this is a decoder for a DCF77 signal.
the decoder decodes the DCF77 signal and checks for a valid Date_Time.
since the dcf77 signal is only secured with a simple parity the decoder waits for two consecutive valid transmissions before it sets the output signals.
given a valid reception by the receiver the decoder can take up to 3 minutes to start its clocks the first time.
after a valid signal is detected the error output goes low and dignals a valid dcf signal from the receiver.
a tp is only valid for one program cycle to allow for external rtc setting.
after a valid signal is detected two independent internal clocks are started (RTC and RTC1), the seconds  of these clocks are generated by software since the dcf signal is only valid for minutes.
rtc is always utc ( world time) and rtc1 can be set to any time zone by setting the time_zone_offset and enabling dst for automatic summertime.
a sync output signals the the rtc and rtc1 are in sync with the dcf77 signal, if the dcf77 signal is lost for more then the sync time the sync output goes low
but the rtc and rtc1 outputs keep running based on software timing until a valid dcf77 signal is received again and triggers the clock.
in addition a millisecond output gives further resolutionof the clocks.
a dst output shows if daylight saving time is enables and the weekday output shows which day of week currently is ( 1= monday ... 7= sunday).


*)
(* if tp was set it should only be active for 1 cycle *)
TP := FALSE;

(* read system time *)
t1 := DWORD_TO_TIME(T_PLC_MS());
tx := t1 - last;

IF rec XOR edge THEN
	edge := rec;
	IF NOT rec AND tx > t#1700ms AND tx < t#2000ms THEN
		(* start condition reached *)
		state := 0;
		tp := NOT error;
	ELSIF NOT rec AND tx > t#700ms AND tx < t#1000ms THEN
		(* second switch detected *)
		IF state < 58 THEN state := state +1; ELSE state := 0; END_IF;
	ELSIF rec AND tx  < t#120ms THEN
		(* bit 0 detected  *)
		bits[state] := 0;
	ELSIF rec AND tx > t#120ms AND tx < t#250ms THEN
		(* bit 1 detected *)
		bits[state] := 1;
	ELSE
		(* error condition received signal is not valid *)
		error := TRUE;
		state := 0;
	END_IF;
	last := last + tx;
	IF rec AND state = 58 THEN
		error := FALSE;

		(* decode the bits and check for possible errors *)
		IF bits[0] OR NOT (bits[17] XOR bits[18]) OR NOT bits[20] THEN error := TRUE; END_IF;
		(* decode minute *)
		minute := 0;
		minute.0 := bits[21];
		minute.1 := bits[22];
		minute.2 := bits[23];
		minute.3 := bits[24];
		IF bits[25] THEN minute := minute + 10; END_IF;
		IF bits[26] THEN minute := minute +20; END_IF;
		IF bits[27] THEN minute := minute +40; END_IF;
		IF minute > 59 OR (bits[21] XOR bits[22] XOR bits[23] XOR bits[24] XOR bits[25] XOR bits[26] XOR bits[27] XOR bits[28]) THEN error := TRUE; END_IF;

		(* decode hour *)
		hour := 0;
		hour.0 := bits[29];
		hour.1 := bits[30];
		hour.2 := bits[31];
		hour.3 := bits[32];
		IF bits[33] THEN hour := hour + 10; END_IF;
		IF bits[34] THEN hour := hour +20; END_IF;
		IF hour > 23 OR (bits[29] XOR bits[30] XOR bits[31] XOR bits[32] XOR bits[33] XOR bits[34] XOR bits[35]) THEN error := TRUE; END_IF;

		(* decode day of month *)
		day := 0;
		day.0 := bits[36];
		day.1 := bits[37];
		day.2 := bits[38];
		day.3 := bits[39];
		IF bits[40] THEN day := day + 10; END_IF;
		IF bits[41] THEN day := day + 20; END_IF;
		IF day > 31 THEN error := TRUE; END_IF;

		(* decode day of week *)
		weekday := 0;
		weekday.0 := bits[42];
		weekday.1 := bits[43];
		weekday.2 := bits[44];
		IF weekday > 7 OR weekday < 1 THEN error := TRUE; END_IF;

		(* decode month *)
		month := 0;
		month.0 := bits[45];
		month.1 := bits[46];
		month.2 := bits[47];
		month.3 := bits[48];
		IF bits[49] THEN month := month +10; END_IF;
		IF month > 12 THEN error := TRUE; END_IF;

		(* decode year *)
		year := 0;
		year.0 := bits[50];
		year.1 := bits[51];
		year.2 := bits[52];
		year.3 := bits[53];
		IF bits[54] THEN year := year + 10; END_IF;
		IF bits[55] THEN year := year + 20; END_IF;
		IF bits[56] THEN year := year + 40; END_IF;
		IF bits[57] THEN year := year + 80; END_IF;

		(* check parity for bits 36 to 58 *)
		cnt := 0;
		FOR i := 36 TO 58 DO IF bits[i] THEN cnt := cnt + 1; END_IF; END_FOR;
		IF NOT even(cnt) THEN error := TRUE; END_IF;

		(* time must be valid for two cycles to clear error flag *)
		IF NOT error THEN
			(* set outputs *)
			old_time := mez;
			IF year >= 70 THEN year := year + 1900; ELSE year := year + 2000; END_IF;
			mez := set_DT(year,month,day,hour,minute,0);
			DST := bits[17];
			IF DST THEN
				UTC := DWORD_TO_DT(DT_TO_DWORD(mez) - 7200);
			ELSE
				UTC := DWORD_TO_DT(DT_TO_DWORD(mez) - 3600);
			END_IF

			(* set trigger signal only if the receiver has received 2 successive minutes *)
			IF mez <> old_time + t#1m THEN error := TRUE ; END_IF;
		END_IF;
	END_IF;
END_IF;

(* this portion implements a free running clock which is triggered by the dcf77 signal *)
IF tp THEN
	rtc := utc;
	IF DST AND dst_en THEN
		IF time_offset < 0 THEN	rtc1 := rtc - INT_TO_TIME(-time_offset) + t#1h; ELSE rtc1 := rtc + INT_TO_TIME(time_offset) + t#1h; END_IF;
	ELSE
		IF time_offset < 0 THEN rtc1 := rtc - INT_TO_TIME(-time_offset); ELSE rtc1 := rtc + INT_TO_TIME(time_offset); END_IF;
	END_IF;
	sync := TRUE;
	last_sync := last;
	ty := last;
ELSIF rtc > DWORD_TO_DT(0) AND T1 - ty >= t#1s THEN
	rtc := rtc + t#1s;
	rtc1 := rtc1 + t#1s;
	ty := ty + t#1s;
	sync := ty - last_sync < sync_timeout AND last_sync > DWORD_TO_TIME(0);
	weekday := weekday(DT_TO_DATE(rtc1));
	DST := dst_en AND DST(utc);
END_IF;
msec := TIME_TO_INT(t1 - ty);



(* decode information
bits		content
0			Bitwert immer 0
1 bis 14	reserviert für Betriebsinformationen (nicht für DCF77-Nutzer bestimmt)
15			Rufbit für Alarmierung der PTB-Mitarbeiter
			(bis Mai 2003: Bitwert = 0 falls normale Antenne in Verwendung; 1 = Backupantenne)
16			Bitwert = 1 falls ein Wechsel von MEZ nach MESZ oder umgekehrt bevorsteht; Dauer der Anzeige: 1 Stunde
17 + 18	gültige Zeit = MEZ, falls Bit 17=0 und Bit 18=1
			gültige Zeit = MESZ, falls Bit 17=1 und Bit 18=0
19			Bitwert = 1 falls innerhalb den nächsten 59 Minuten eine Schaltsekunde angeordnet ist. Beim Einfügen einer Schaltsekunde wird anstelle der 59. die 60. Sekundenmarke weggelassen und in der 58. erfolgt ausnahmsweise ein Trägerabfall.
20			Startbit für Zeitinformation (immer 1)
21 - 27		1, 2, 4, 8, 10, 20, 40 Minuten (bitweise Addition)
28			Prüfbit (gerade Parität) für die Bits 21-27
29 - 34		1, 2, 4, 8, 10, 20 Stunden (bitweise Addition)
35			Prüfbit (gerade Parität) für die Bits 29-34
36 - 41		Tagesnummer im aktuellen Monat: 1, 2, 4, 8, 10, 20 (bitweise Addition)
42 - 44		Tagesnummer in der aktuellen Woche: 1, 2, 4 (bitweise Addition)
45 - 49		Monatsnummer: 1, 2, 4, 8, 10 (bitweise Addition)
50 - 57		Jahr (zweistellig): 1, 2, 4, 8, 10, 20, 40, 80 (bitweise Addition)
58			Prüfbit (gerade Parität) füR die Bits 36-57

*)
(* revision history

hm 2.feb 2007		rev 1.1
	change wday and dst outputs when there is no dcf reception

hm	26.feb 2007		rev 1.2
	changed statements where t#1h would be substracted from DT.
	under certain conditions the compiler would crash translating this statement

hm	17. sep 2007	rev 1.3
	replaced time() with T_PLC_MS() for compatibility reasons

hm	24. oct 2007	rev 1.4
	changed dst calculation because function dst was upgraded no error in DCF77 only a change in DST

hm	12. nov 2007	rev 1.5
	changed time_offset from time to integer to allow for negative offset time zones

*)
END_FUNCTION_BLOCK

(* POU Time&Date/DST, ST *)
FUNCTION DST : BOOL
VAR_INPUT
	utc : DT;
END_VAR
VAR
	yr : INT;
	yr4 : DWORD;
	ltc: DWORD;
	idate : DWORD;
END_VAR

(*
version 1.1	24 oct 2007
programmer 	hugo
tested by		tobias

this functions returns TRUE IF dst TIME is active 
the FUNCTION calculates automatically for any year betweek 1970 AND 2099 
wheather daylight savings is on OR off 
the summertime calculation is done according to european standards.
dst will become TRUE AT 01:00 utc in the morning FOR the respective days 
AND it will become FALSE after daylight savings TIME is switched back end OF october at 01:00 utc

*)
yr := year(DT_TO_DATE(utc));
ltc := DT_TO_DWORD(utc);
idate := DT_TO_DWORD(set_DT(yr,3,31,1,0,0));
yr4 := 5*yr/4;
IF idate - ((yr4+4) MOD 7)*86400 <= ltc AND idate + (214 - (yr4+1) MOD 7)*86400 > ltc THEN DST := TRUE; ELSE DST := FALSE; END_IF;

(* revision history
hm	4. aug 2006		rev 1.0
	original version

hm	24. okt 2007	rev 1.1
	deleted time_zone_offset input because dst is generally at 01:00 utc and not mesz
	uk starts 01:00 utc and also greece

*)

(*
Equation used TO calculate the beginning OF European Summer TIME:
Sunday (31 - (5*y/4 + 4) mod 7) March at 01.00 UTC
(valid through 2099, courtesy of Robert H. van Gent, EC).

European Summer Time ends (clocks go back) at 01.00 UTC on

    * 29 October 2006
    * 28 October 2007
    * 26 October 2008

Equation used to calculate the end of European Summer Time:
Sunday (31 - (5*y/4 + 1) mod 7) October at 01.00 UTC
(validity AND credits as above).

*)
END_FUNCTION

(* POU engineering/control/dead_zone, ST *)
FUNCTION dead_zone : REAL
VAR_INPUT
	X : REAL;
	L : REAL;
END_VAR
VAR
END_VAR

(*
version 1.0	12 Feb 2007
programmer 	hugo
tested by		tobias

dead_zone2 is a linear transfer function which follows a linear function except for x is close to 0.
Y = X if abs(x) > L otherwise its 0.

*)
IF ABS(x) > L THEN
	dead_zone := X;
ELSE
	dead_zone := 0;
END_IF;
END_FUNCTION

(* POU engineering/control/dead_zone2, ST *)
FUNCTION_BLOCK dead_zone2
VAR_INPUT
	X : REAL;
	L : REAL;
END_VAR
VAR_OUTPUT
	Y: REAL;
END_VAR
VAR
END_VAR

(*
version 1.0	12 Feb 2007
programmer 	hugo
tested by		tobias

dead_zone2 is a linear transfer function which follows a linear function except for x is close to 0.
Y = X if abs(x) > L.
for values of 0 +/. L a hysteresis function will hold the output at + or - L.

*)
IF ABS(x) > L THEN
	Y := X;
ELSIF Y > 0 THEN
	Y := L;
ELSE
	Y := -L;
END_IF;
END_FUNCTION_BLOCK

(* POU Logic/gate logic/DEC_2, ST *)
FUNCTION_BLOCK DEC_2
VAR_INPUT
	D: BOOL;
	A: BOOL;
END_VAR
VAR_OUTPUT
	Q0: BOOL;
	Q1: BOOL;
END_VAR
VAR
END_VAR

(*
version 1.1	3 Mar 2007
programmer 	hugo
tested by		tobias

a bit input will be decoded to the two outputs Q0 or Q1
dependent on the value of A
A=0 decodes to Q0 and A=1 decodes to Q1

*)
Q0 := D AND NOT A;
Q1 := D AND A;

(* revision history
hm 3.3.2007	rev 1.1
	rewritten in ST for better compatibility

*)
END_FUNCTION_BLOCK

(* POU Logic/gate logic/DEC_4, ST *)
FUNCTION_BLOCK DEC_4
VAR_INPUT
	D: BOOL;
	A0: BOOL;
	A1: BOOL;
END_VAR
VAR_OUTPUT
	Q0: BOOL;
	Q1: BOOL;
	Q2: BOOL;
	Q3: BOOL;
END_VAR
VAR
END_VAR

(*
version 1.1	3 Mar 2007
programmer 	hugo
tested by		tobias

a bit input will be decoded to one of the 4 outputs
dependent on the Adress on A0 and A1

executioin TIME on wago 750-841 = 9us
*)
Q0 := D AND NOT A0 AND NOT A1;
Q1 := D AND A0 AND NOT A1;
Q2 := D AND NOT A0 AND A1;
Q3 := D AND A0 AND A1;

(* revision history
hm 3.3.2007	rev 1.1
	rewritten in ST for better compatibility

*)
END_FUNCTION_BLOCK

(* POU Logic/gate logic/DEC_8, ST *)
FUNCTION_BLOCK DEC_8
VAR_INPUT
	D: BOOL;
	A0: BOOL;
	A1: BOOL;
	A2: BOOL;
END_VAR
VAR_OUTPUT
	Q0: BOOL;
	Q1: BOOL;
	Q2: BOOL;
	Q3: BOOL;
	Q4: BOOL;
	Q5: BOOL;
	Q6: BOOL;
	Q7: BOOL;
END_VAR
VAR
END_VAR

(*
version 1.1	3 mar 2007
programmer 	hugo
tested by		tobias

a bit input will be decoded to one of the 8 outputs
dependent on the Adress on A0, A1 and A2

executioin TIME on wago 750-841 = 17us
*)
Q0 := D AND NOT A0 AND NOT A1 AND NOT A2;
Q1 := D AND A0 AND NOT A1 AND NOT A2;
Q2 := D AND NOT A0 AND A1 AND NOT A2;
Q3 := D AND A0 AND A1 AND NOT A2;
Q4 := D AND NOT A0 AND NOT A1 AND A2;
Q5 := D AND A0 AND NOT A1 AND A2;
Q6 := D AND NOT A0 AND A1 AND A2;
Q7 := D AND A0 AND A1 AND A2;

(* revision history
hm 3.3.2007	rev 1.1
	rewritten in ST for better compatibility

*)
END_FUNCTION_BLOCK

(* POU engineering/signal processing/delay, ST *)
FUNCTION_BLOCK delay
VAR_INPUT
	in : REAL;
	N : INT;
	rst : BOOL;
END_VAR
VAR_OUTPUT
	out : REAL;
END_VAR
VAR
	buf : ARRAY[0..31] OF REAL;
	i : INT;
END_VAR

(*
version 1.2	19. jan 2007
programmer 	hugo
tested by		tobias

this function block delays input values by each programm cycle
after N+1 cycles the in value has shifted to the out.
N can be any alue from 0 .. 32
if n = 0 the input will be present on the output without a delay.
f N > 32 then the output will be delayed by 32 cycles.
any high on rst will load the buffer with in.

*)
IF N > SIZEOF(buf) / SIZEOF(in) THEN N:= 32; END_IF;
IF rst THEN
	FOR i := 0 TO 31 DO buf[i] := 0; END_FOR;
	out := in;
ELSIF N < 1 THEN out := in;
ELSE
	IF i >= N THEN i := 0; END_IF;
	out := buf[i];
	buf[i] := in;
	i := i + 1;
END_IF;

(* revision history
hm 1.10.2006	rev 1.1
	corrected error in buffer management

hm 19.1.2007	rev 1.2
	changed reset to load the value of in instead of 0

*)
END_FUNCTION_BLOCK

(* POU engineering/signal processing/delay_4, ST *)
FUNCTION_BLOCK delay_4
VAR_INPUT
	in : REAL;
END_VAR
VAR_OUTPUT
	out1 : REAL;
	out2 : REAL;
	out3 : REAL;
	out4 : REAL;
END_VAR
VAR
	temp: REAL;
END_VAR

(*
version 1.1	19 jan 2007
programmer 	hugo
tested by		tobias

this function block delays input values by each programm cycle
after 4 cycles the in value has shifted to the out 4 and will be discarded after the next cycle
the blocks can be cascaded.

*)
out4 := out3;
out3 := out2;
out2 := out1;
out1 := temp;
temp := in;

(* revision history

hm 19.1.2007	rev 1.1
	added variable temp to add 1 delay  for q1

*)
END_FUNCTION_BLOCK

(* POU Building/electrical/dimm_i, ST *)
FUNCTION_BLOCK dimm_i
VAR_INPUT
	set : BOOL;
	in : BOOL;
	rst : BOOL;
END_VAR
VAR_INPUT CONSTANT
	T_debounce : TIME := T#10ms;
	T_reconfig : TIME := T#10s;
	T_on_max : TIME := T#0h;
	T_dimm_start : TIME := T#1s;
	T_dimm: TIME := T#3s;
END_VAR
VAR_OUTPUT
	Q : BOOL := 0;
	out : BYTE := 0;
END_VAR
VAR
	tx : TIME := T#0s;
	last_edge : BOOL;
	state : BYTE := 0;
	edge : BOOL := 0;
	r_edge : BOOL := 0;
	T_on : TIME;
	dimm_up: BOOL;
	last_step : TIME;
	tn: TIME;
END_VAR

(*
version 1.3	15 sep 2007
programmer 	hugo
tested by		tobias

this is an intelligent dimmer interface with an autoset feature for "in" it will automatically detect the type of switch:
low active pulses or high high active pulses are allowd for in.
a configurable debounce timer will debounce input signals
if t_on_max is set to anything other then 0 the output will be turned off after the max on time is reached.
the times for debounce, dimming ramp, wait time before dimming and max on time are all programmable.

the dimmer has outputs Q for on and off and also out with the analog dimm value.

*)
(* read system time *)
tn := DWORD_TO_TIME(T_PLC_MS());;

IF rst THEN
	state := 0;
	Q := 0;
	dimm_up := TRUE;
ELSIF set THEN
	state := 0;
	Q := TRUE;
	out := 255;
	dimm_up := FALSE;
	T_on := Tn;
ELSE
	CASE state OF
	(* state 0 wait for activity *)
	0 :	IF (r_edge AND in AND NOT edge) OR (NOT r_edge AND NOT in AND edge) THEN
			IF t_debounce = t#0s THEN state := 2;  ELSE state := 1; END_IF;
			tx := Tn;
			last_edge := in;
		END_IF

	(* state 1 debouncing *)
	1:	IF Tn - T_debounce >= tx THEN
			state := 2;
			tx := Tn;
		END_IF;

	(* state 2 wait for second edge to toggle output *)
	2:	IF Tn - T_dimm_start >= tx THEN
			state := 3;
			tx := Tn;
			(* time to switch elapsed without switching if Q = 0 turn on output and start dimming at 1 *)
			IF NOT Q THEN
				Q := TRUE;
				t_on := tx;
				out := 1;
				dimm_up := TRUE;
			ELSE
				IF out =255 THEN dimm_up := FALSE; END_IF;
			END_IF;
		ELSIF in XOR edge THEN
			(* wait for edge to toggle output and stop all activity *)
			IF Q THEN
				Q := FALSE;
				state := 0;
			ELSE
				Q := TRUE;
				state := 3;
				IF out = 0 THEN out := 255; END_IF
				IF out = 255 THEN dimm_up := FALSE; END_IF;
				tx := Tn;
				t_on := tx;
			END_IF;
		END_IF;

	(* state 3 entered dimming phase *)
	3:	IF in AND r_edge THEN
			(* generate ramp *)
			tx := Tn;
			IF tx >= last_step + T_dimm / 255 THEN
				last_step := tx;
				IF dimm_up AND out < 255 THEN
					out := out + 1;
					IF out = 255 THEN
						dimm_up := FALSE;
						state := 0;
					END_IF;
				ELSIF NOT dimm_up AND out > 0 THEN
					out := out -1;
					IF out = 0 THEN
						Q := FALSE;
						state := 0;
						dimm_up := TRUE;
					 END_IF;
				 END_IF;
			END_IF;
		ELSE
			dimm_up := NOT dimm_up;
			state := 0;
		END_IF;

	END_CASE;

	(* check for max t_on time and reset output if too long *)
	IF Q AND t_on_max > T#0s AND Tn - t_on_max >= T_on THEN Q := 0; END_IF;

	(* check for reconfig and set R_edge to high for rising edge sensitivity *)
	IF Tn - T_reconfig >= tx THEN R_edge := NOT in; END_IF;

	(* set edge to follow in for next edge detection *)
	edge := in;
END_IF;


(* revision history

hm 22.1.2007		rev 1.1
	deleted unused structure ramp

hm 2.feb 2007		rev 1.2
	changed structure to read time() at the beginning for better time consistency if a higher priorized tak interrupts dimm_i
	added statements in case structure for state 1 to allow for short 1 cycle input pulses

hm 	15.9.2007		rev 1.3
	replaced Time() with T_PLC_MS for compatibility and performance reasons

*)
END_FUNCTION_BLOCK

(* POU Logic/gate logic/DWord_of_Byte, ST *)
FUNCTION DWord_of_Byte : DWORD
VAR_INPUT
	B0 : BYTE;
	B1 : BYTE;
	B2 : BYTE;
	B3 : BYTE;
END_VAR
VAR
END_VAR

(*
version 1.0	24 jan 2007
programmer 	hugo
tested by		tobias

this function creates a Dword from 4 individual bytes

*)
DWord_of_Byte := B3;
DWord_of_Byte := SHL(DWord_of_Byte,8) OR B2;
DWord_of_Byte := SHL(DWord_of_Byte,8) OR B1;
DWord_of_Byte := SHL(DWord_of_Byte,8) OR B0;
END_FUNCTION

(* POU String/DWORD_To_STRF, ST *)
FUNCTION DWORD_To_STRF : STRING
VAR_INPUT
	IN : DWORD;
	N : INT;
END_VAR
VAR
	L: INT;
	temp: STRING;
END_VAR

(*
version 1.0	26 jan 2007
programmer 	hugo
tested by		tobias

dword_to_strF converts a DWORD, BYTE or Word to a fixed length String.
the string will be filles with leading zeroes to achieve the fixed length, or if too long, the lowest digits will be used.

for example:	dword_to_strf(123,4) = '0123' 
				dword_to_strf(123,2) = '23'
*)
(* convert dword to string first and cut to length N *)
temp := RIGHT(DWORD_TO_STRING(in),N);
L := LEN(temp);
WHILE L < N DO
	temp := CONCAT('0', temp);
	L := L + 1;
END_WHILE;
DWORD_To_STRF := temp;
END_FUNCTION

(* POU mathematical/Geometry/ellipse_A, ST *)
FUNCTION ellipse_A : REAL
VAR_INPUT
	R1 : REAL;
	R2 : REAL;
END_VAR
VAR
END_VAR

(*
version 1.0	16 oct 2007
programmer 	hugo
tested by		tobias

ellipse_A calculates the Area of an ellipe based on the two radians R1 and R2


*)
ellipse_A := PI1 * R1 * R2;

(* revision histroy
hm	16. oct 2007	rev 1.0
	original version

*)
END_FUNCTION

(* POU mathematical/Geometry/ellipse_C, ST *)
FUNCTION ellipse_C : REAL
VAR_INPUT
	R1 : REAL;
	R2 : REAL;
END_VAR
VAR
END_VAR

(*
version 1.0	16 oct 2007
programmer 	hugo
tested by		tobias

ellipse_C calculates the circumference of an ellipe based on the two radians R1 and R2

*)
ellipse_C := PI1 * (3*(R1+R2) - SQRT((3*r1 + R2)*(3*r2 + r1)));

(* revision histroy
hm	16. oct 2007	rev 1.0
	original version

*)
END_FUNCTION

(* POU engineering/conversion/energy, ST *)
FUNCTION_BLOCK energy
VAR_INPUT
	J : REAL;
	C : REAL;
	Wh : REAL;
END_VAR
VAR_OUTPUT
	YJ : REAL;
	YC : REAL;
	YWh : REAL;
END_VAR
VAR
END_VAR

(*
version 1.0	27 mar 2007
programmer 	hugo
tested by		oscat

this function converts different energy units
any unused input can simply be left open.
different inputs connected at the same time will be added up.
*)
YJ := J + Wh * 3600 + C * 4.1868;
YC := YJ / 4.1868;
YWh := YJ / 3600;

(*
Arbeit, Energie, Joule* J 1 J = 1 N · m = 1 W · s = (1/3,6) E–6 kW · h = 1 kg · m2/s2
Wärmemenge Kilowattstunde kW · h 1 kW · h = 3,6 MJ = 860 kcal
Elektronvolt eV 1 eV = 160,218 92 E–21 J
Erg erg 1 erg = 1E–7 J
Kalorie cal 1 cal = 4,1868 J = 1,163 E–3 W · h
Therm therm 1 therm = 105,50 · 106 J

*)
END_FUNCTION_BLOCK

(* POU other/ESR_collect, ST *)
FUNCTION_BLOCK ESR_collect
VAR_INPUT
	ESR_0, ESR_1, ESR_2, ESR_3, ESR_4, ESR_5, ESR_6, ESR_7 : ARRAY [0..3] OF esr_data;
END_VAR
VAR_OUTPUT
	ESR_OUT : ARRAY[0..63] OF esr_data;
	pos : INT;
END_VAR
VAR CONSTANT
	max_in : INT := 3; (* maximum element of input variable *)
	max_out : INT := 63; (* maximum element of output array *)
END_VAR
VAR
	cnt : INT;
END_VAR

(*
version 1.0	26 jan 2007
programmer 	hugo
tested by		tobias

ESR_collect collects esr data from up to 8 esr_mon modules and stroes them in an output array.
the output pos will display the position of the last element in the array.
if the array will be full, the oldest element is overwritten.

*)
FOR cnt := 0 TO max_in DO
	IF esr_0[cnt].typ > 0 THEN
		esr_out[pos] := esr_0[cnt];
		pos := pos + 1;
		IF pos > max_out THEN pos := 0; END_IF;
	END_IF;
END_FOR;
FOR cnt := 0 TO max_in DO
	IF esr_1[cnt].typ > 0 THEN
		esr_out[pos] := esr_1[cnt];
		pos := pos + 1;
		IF pos > max_out THEN pos := 0; END_IF;
	END_IF;
END_FOR;
FOR cnt := 0 TO max_in DO
	IF esr_2[cnt].typ > 0 THEN
		esr_out[pos] := esr_2[cnt];
		pos := pos + 1;
		IF pos > max_out THEN pos := 0; END_IF;
	END_IF;
END_FOR;
FOR cnt := 0 TO max_in DO
	IF esr_3[cnt].typ > 0 THEN
		esr_out[pos] := esr_3[cnt];
		pos := pos + 1;
		IF pos > max_out THEN pos := 0; END_IF;
	END_IF;
END_FOR;
FOR cnt := 0 TO max_in DO
	IF esr_4[cnt].typ > 0 THEN
		esr_out[pos] := esr_4[cnt];
		pos := pos + 1;
		IF pos > max_out THEN pos := 0; END_IF;
	END_IF;
END_FOR;
FOR cnt := 0 TO max_in DO
	IF esr_5[cnt].typ > 0 THEN
		esr_out[pos] := esr_5[cnt];
		pos := pos + 1;
		IF pos > max_out THEN pos := 0; END_IF;
	END_IF;
END_FOR;
FOR cnt := 0 TO max_in DO
	IF esr_6[cnt].typ > 0 THEN
		esr_out[pos] := esr_6[cnt];
		pos := pos + 1;
		IF pos > max_out THEN pos := 0; END_IF;
	END_IF;
END_FOR;
FOR cnt := 0 TO max_in DO
	IF esr_7[cnt].typ > 0 THEN
		esr_out[pos] := esr_7[cnt];
		pos := pos + 1;
		IF pos > max_out THEN pos := 0; END_IF;
	END_IF;
END_FOR;
END_FUNCTION_BLOCK

(* POU other/ESR_MON_B8, ST *)
FUNCTION_BLOCK ESR_MON_B8
VAR_INPUT
	s0, s1, s2, s3, s4, s5, s6, s7 : BOOL;
	DT_in : DT;
END_VAR
VAR_INPUT CONSTANT
	a0, a1, a2, a3, a4, a5, a6, a7 : STRING(10);
END_VAR
VAR_OUTPUT
	ESR_Out: ARRAY [0..3] OF esr_data;
	ESR_Flag : BOOL;
END_VAR
VAR
	x0, x1, x2, x3, x4, x5, x6, x7 : BOOL;
	tx: TIME;
	cnt : INT;
END_VAR

(*
version 1.1	17 sep 2007
programmer 	hugo
tested by		tobias

ESR_mon_B8 monitores up to 8 binary inputs and reports changes with time stamd and adress label.
the module checks 8 inputs for a change and reports all changes with time and adress stamp to the output.
4 events maximum can be collected at once within the same cycle

*)
(* read system timer *)
tx := DWORD_TO_TIME(T_PLC_MS());

ESR_Flag := FALSE;
esr_out[3].typ := 0;
esr_out[2].typ := 0;
esr_out[1].typ := 0;
esr_out[0].typ := 0;
cnt := 0;

(* check if inputs have chaged and fill buffer *)
IF s0 <> X0 THEN
	IF s0 THEN esr_out[cnt].typ := 11; ELSE 	esr_out[cnt].typ := 10; END_IF;
	esr_out[cnt].adress := a0;
	esr_out[cnt].DS := DT_in;
	esr_out[cnt].TS := TX;
	X0 := S0;
	cnt := cnt + 1;
	esr_flag := TRUE;
END_IF;
IF s1 <> X1 THEN
	IF s1 THEN esr_out[cnt].typ := 11; ELSE 	esr_out[cnt].typ := 10; END_IF;
	esr_out[cnt].adress := a1;
	esr_out[cnt].DS := DT_in;
	esr_out[cnt].TS := TX;
	X1 := S1;
	cnt := cnt + 1;
	esr_flag := TRUE;
END_IF;
IF s2 <> X2 THEN
	IF s2 THEN esr_out[cnt].typ := 11; ELSE 	esr_out[cnt].typ := 10; END_IF;
	esr_out[cnt].adress := a2;
	esr_out[cnt].DS := DT_in;
	esr_out[cnt].TS := TX;
	X2 := S2;
	cnt := cnt + 1;
	esr_flag := TRUE;
END_IF;
IF s3 <> X3 THEN
	IF s3 THEN esr_out[cnt].typ := 11; ELSE 	esr_out[cnt].typ := 10; END_IF;
	esr_out[cnt].adress := a3;
	esr_out[cnt].DS := DT_in;
	esr_out[cnt].TS := TX;
	X3 := S3;
	cnt := cnt + 1;
	esr_flag := TRUE;
END_IF;
IF s4 <> X4 AND cnt < 4 THEN
	IF s4 THEN esr_out[cnt].typ := 11; ELSE 	esr_out[cnt].typ := 10; END_IF;
	esr_out[cnt].adress := a4;
	esr_out[cnt].DS := DT_in;
	esr_out[cnt].TS := TX;
	X4 := S4;
	cnt := cnt + 1;
	esr_flag := TRUE;
END_IF;
IF s5 <> X5  AND cnt < 4 THEN
	IF s5 THEN esr_out[cnt].typ := 11; ELSE 	esr_out[cnt].typ := 10; END_IF;
	esr_out[cnt].adress := a5;
	esr_out[cnt].DS := DT_in;
	esr_out[cnt].TS := TX;
	X5 := S5;
	cnt := cnt + 1;
	esr_flag := TRUE;
END_IF;
IF s6 <> X6  AND cnt < 4 THEN
	IF s6 THEN esr_out[cnt].typ := 11; ELSE 	esr_out[cnt].typ := 10; END_IF;
	esr_out[cnt].adress := a6;
	esr_out[cnt].DS := DT_in;
	esr_out[cnt].TS := TX;
	X6 := S6;
	cnt := cnt + 1;
	esr_flag := TRUE;
END_IF;
IF s7 <> X7  AND cnt < 4 THEN
	IF s7 THEN esr_out[cnt].typ := 11; ELSE 	esr_out[cnt].typ := 10; END_IF;
	esr_out[cnt].adress := a7;
	esr_out[cnt].DS := DT_in;
	esr_out[cnt].TS := TX;
	X7 := S7;
	cnt := cnt + 1;
	esr_flag := TRUE;
END_IF;

(* revision history
hm	26. jan 2007		rev 1.0
	original version

hm	17. sep 2007	rev 1.1
	replaced time() with T_PLC_MS() for compatibility reasons
	
*)
END_FUNCTION_BLOCK

(* POU other/ESR_MON_R4, ST *)
FUNCTION_BLOCK ESR_MON_R4
VAR_INPUT
	R0, R1, R2, R3 : REAL;
	DT_in : DT;
END_VAR
VAR_INPUT CONSTANT
	a0, a1, a2, a3 : STRING(10);
	s0, s1, s2, s3 : REAL;
END_VAR
VAR_OUTPUT
	ESR_Out: ARRAY [0..3] OF esr_data;
	ESR_Flag : BOOL;
END_VAR
VAR
	x0, x1, x2, x3 : REAL;
	tx: TIME;
	cnt : INT;
END_VAR

(*
version 1.1 17 sep 2007
programmer 	hugo
tested by		tobias

ESR_mon_R4 monitores up to 4 Real inputs and reports changes with time stamd and adress label.
the module checks 4 inputs for a change of more than the specified sensitivity S and reports all changes with time and adress stamp to the output.

*)
(* read system timer *)
tx := DWORD_TO_TIME(T_PLC_MS());

ESR_Flag := FALSE;
esr_out[3].typ := 0;
esr_out[2].typ := 0;
esr_out[1].typ := 0;
esr_out[0].typ := 0;
cnt := 0;

(* check if inputs have chaged and fill buffer *)
IF differ(R0,  X0, S0) THEN
	esr_out[cnt].adress := a0;
	esr_out[cnt].DS := DT_in;
	esr_out[cnt].TS := TX;
	esr_out[cnt].data[0] := REAL_TO_BYTE(R0);
	esr_out[cnt].data[1] := DWORD_TO_BYTE(SHR(REAL_TO_DWORD(R0),8));
	esr_out[cnt].data[2] := DWORD_TO_BYTE(SHR(REAL_TO_DWORD(R0),16));
	esr_out[cnt].data[3] := DWORD_TO_BYTE(SHR(REAL_TO_DWORD(R0),24));
	X0 := R0;
	cnt := cnt + 1;
	esr_flag := TRUE;
END_IF;
IF differ(R1,  X1, S1) THEN
	esr_out[cnt].adress := a1;
	esr_out[cnt].DS := DT_in;
	esr_out[cnt].TS := TX;
	esr_out[cnt].data[0] := REAL_TO_BYTE(R1);
	esr_out[cnt].data[1] := DWORD_TO_BYTE(SHR(REAL_TO_DWORD(R1),8));
	esr_out[cnt].data[2] := DWORD_TO_BYTE(SHR(REAL_TO_DWORD(R1),16));
	esr_out[cnt].data[3] := DWORD_TO_BYTE(SHR(REAL_TO_DWORD(R1),24));
	X1 := R1;
	cnt := cnt + 1;
	esr_flag := TRUE;
END_IF;
IF differ(R2,  X2, S2) THEN
	esr_out[cnt].adress := a2;
	esr_out[cnt].DS := DT_in;
	esr_out[cnt].TS := TX;
	esr_out[cnt].data[0] := REAL_TO_BYTE(R2);
	esr_out[cnt].data[1] := DWORD_TO_BYTE(SHR(REAL_TO_DWORD(R2),8));
	esr_out[cnt].data[2] := DWORD_TO_BYTE(SHR(REAL_TO_DWORD(R2),16));
	esr_out[cnt].data[3] := DWORD_TO_BYTE(SHR(REAL_TO_DWORD(R2),24));
	X2 := R2;
	cnt := cnt + 1;
	esr_flag := TRUE;
END_IF;
IF differ(R3,  X3, S3) THEN
	esr_out[cnt].adress := a3;
	esr_out[cnt].DS := DT_in;
	esr_out[cnt].TS := TX;
	esr_out[cnt].data[0] := REAL_TO_BYTE(R3);
	esr_out[cnt].data[1] := DWORD_TO_BYTE(SHR(REAL_TO_DWORD(R3),8));
	esr_out[cnt].data[2] := DWORD_TO_BYTE(SHR(REAL_TO_DWORD(R3),16));
	esr_out[cnt].data[3] := DWORD_TO_BYTE(SHR(REAL_TO_DWORD(R3),24));
	X3 := R3;
	cnt := cnt + 1;
	esr_flag := TRUE;
END_IF;


(* revision history
hm	26. jan 2007		rev 1.0
	original version

hm	17. sep 2007	rev 1.1
	replaced time() with T_PLC_MS() for compatibility reasons
	
*)
END_FUNCTION_BLOCK

(* POU other/ESR_MON_X8, ST *)
FUNCTION_BLOCK ESR_MON_X8
VAR_INPUT
	s0, s1, s2, s3, s4, s5, s6, s7 : BYTE;
	DT_in : DT;
	Mode : BYTE := 3;
END_VAR
VAR_INPUT CONSTANT
	a0, a1, a2, a3, a4, a5, a6, a7 : STRING(10);
END_VAR
VAR_OUTPUT
	ESR_Out: ARRAY [0..3] OF esr_data;
	ESR_Flag : BOOL;
END_VAR
VAR
	x0, x1, x2, x3, x4, x5, x6, x7 : BYTE;
	tx: TIME;
	cnt : INT;
END_VAR

(*
version 1.1	17 sep 2007
programmer 	hugo
tested by		tobias

ESR_MON_X8 is a status and error collector.
the module checks 8 status inputs for a change and reports up to 4 input changes with time and adress stamp to the output.
the mode can be 
1 for error only
2 for error and status
3 for error, status and debug
the adress label of the 8 inputs can be configured individually.
*)
(* read system timer *)
tx := DWORD_TO_TIME(T_PLC_MS());

ESR_Flag := FALSE;
esr_out[3].typ := 0;
esr_out[2].typ := 0;
esr_out[1].typ := 0;
esr_out[0].typ := 0;
cnt := 0;

(* check if inputs have chaged and fill buffer *)
IF s0 <> X0 AND ((s0 < 100) OR (S0 > 99 AND S0 < 200 AND mode >= 2) OR (S0 > 199 AND mode = 3)) THEN
	esr_out[cnt] := status_to_ESR(s0, a0, DT_in, TX);
	X0 := S0;
	cnt := cnt + 1;
	esr_flag := TRUE;
END_IF;
IF s1 <> X1 AND ((s1 < 100) OR (S1 > 99 AND S1 < 200 AND mode >= 2) OR (S1 > 199 AND mode = 3)) THEN
	esr_out[cnt] := status_to_ESR(s1, a1, DT_in, TX);
	X1 := S1;
	cnt := cnt + 1;
	esr_flag := TRUE;
END_IF;
IF s2 <> X2 AND ((s2 < 100) OR (S2 > 99 AND S2 < 200 AND mode >= 2) OR (S2 > 199 AND mode = 3)) THEN
	esr_out[cnt] := status_to_ESR(s2, a2, DT_in, TX);
	X2 := S2;
	cnt := cnt + 1;
	esr_flag := TRUE;
END_IF;
IF s3 <> X3 AND ((s3 < 100) OR (S3 > 99 AND S3 < 200 AND mode >= 2) OR (S3 > 199 AND mode = 3)) THEN
	esr_out[cnt] := status_to_ESR(s3, a3, DT_in, TX);
	X3 := S3;
	cnt := cnt + 1;
	esr_flag := TRUE;
END_IF;
IF cnt < 4 AND s4 <> X4 AND ((s4 < 100) OR (S4 > 99 AND S4 < 200 AND mode >= 2) OR (S4 > 199 AND mode = 3)) THEN
	esr_out[cnt] := status_to_ESR(s4, a4, DT_in, TX);
	X4 := S4;
	cnt := cnt + 1;
	esr_flag := TRUE;
END_IF;
IF cnt < 4 AND s5 <> X5 AND ((s5 < 100) OR (S5 > 99 AND S5 < 200 AND mode >= 2) OR (S5 > 199 AND mode = 3)) THEN
	esr_out[cnt] := status_to_ESR(s5, a5, DT_in, TX);
	X5 := S5;
	cnt := cnt + 1;
	esr_flag := TRUE;
END_IF;
IF cnt < 4 AND s6 <> X6 AND ((s6 < 100) OR (S6 > 99 AND S6 < 200 AND mode >= 2) OR (S6 > 199 AND mode = 3)) THEN
	esr_out[cnt] := status_to_ESR(s6, a6, DT_in, TX);
	X6 := S6;
	cnt := cnt + 1;
	esr_flag := TRUE;
END_IF;
IF cnt < 4 AND s7 <> X7 AND ((s7 < 100) OR (S7 > 99 AND S7 < 200 AND mode >= 2) OR (S7 > 199 AND mode = 3)) THEN
	esr_out[cnt] := status_to_ESR(s7, a7, DT_in, TX);
	X7 := S7;
	cnt := cnt + 1;
	esr_flag := TRUE;
END_IF;


(* revision history
hm	26. jan 2007		rev 1.0
	original version

hm	17. sep 2007	rev 1.1
	replaced time() with T_PLC_MS() for compatibility reasons
	
*)
END_FUNCTION_BLOCK

(* POU other/status_to_ESR, ST *)
FUNCTION status_to_ESR : esr_data
VAR_INPUT
	status : BYTE;
	adress : STRING(10);
	DT_in : DT;
	TS : TIME;
END_VAR
VAR
END_VAR

(*
version 1.0	6 oct 2006
programmer 	hugo
tested by		tobias

status_to_esr creates esr data from a status byte.

*)
IF status < 100 THEN
	status_to_ESR.typ := 1;
ELSIF status < 200 THEN
	status_to_ESR.typ := 2;
ELSE
	status_to_ESR.typ := 3;
END_IF;
status_to_ESR.adress:= adress;
status_to_ESR.DS := DT_in;
status_to_ESR.TS := TS;
status_to_ESR.data[0] := status;
END_FUNCTION

(* POU String/exec, ST *)
FUNCTION exec : STRING
VAR_INPUT
	str : STRING;
END_VAR
VAR
	pos: INT;
	R1: REAL;
	R2: REAL;
	operator: STRING;
END_VAR

(*
version 1.1	6 feb 2007
programmer 	hugo
tested by		tobias

exec executes a mathematical term and returns the result as a string
the term can only be a simple term without brackets and only one operator
allowed operastors are: (+, -, *, /, ^, sqrt, sin, cos, tan).

*)
(* extract both numbers and operator *)
exec := uppercase(trim(str));

pos := findB_nonum(exec);
IF pos > 1 THEN R1 := STRING_TO_REAL(exec); END_IF;
R2 := STRING_TO_REAL(RIGHT(exec,LEN(exec)-pos));
exec := LEFT(exec,pos);
pos := findB_Num(exec);
operator := RIGHT(exec,LEN(exec) - pos);
IF operator = '' AND LEN(str) = 0 THEN
	exec := '';
	RETURN;
ELSIF operator = '' THEN
	exec := str;
	RETURN;
END_IF;
IF operator = '^' THEN
	exec := REAL_TO_STRING(EXPT(R1, R2));
ELSIF operator = 'SQRT' THEN
	exec := REAL_TO_STRING(SQRT(R2));
ELSIF operator = 'SIN' THEN
	exec := REAL_TO_STRING(SIN(r2));
ELSIF operator = 'COS' THEN
	exec := REAL_TO_STRING(COS(r2));
ELSIF operator = 'TAN' THEN
	exec := REAL_TO_STRING(TAN(R2));
ELSIF operator = '*' THEN
	exec := REAL_TO_STRING(R1 * R2);
ELSIF operator = '/' THEN
	IF R2 <> 0 THEN exec := REAL_TO_STRING(R1 / R2); ELSE exec := 'ERROR'; END_IF;
ELSIF operator = '+' THEN
	exec := REAL_TO_STRING(r1 + r2);
ELSIF operator = '-' THEN
	exec := REAL_TO_STRING(r1 - r2);
ELSE
	exec := 'ERROR';
END_IF;


(* revision history

hm 6.feb 2007	rev 1.1
	cos has to be written in uppercase
	divide by 0 will return an error
     
*)
END_FUNCTION

(* POU String/uppercase, ST *)
FUNCTION uppercase : STRING
VAR_INPUT
	str : STRING;
END_VAR
VAR
	PT : POINTER TO BYTE;
	pos: INT;
END_VAR

(*
version 1.0	6 oct 2006
programmer 	hugo
tested by		tobias

uppercase returns str while all letters a..z are converted to uppercase

*)
PT := ADR(uppercase);
uppercase := str;
FOR pos := 1 TO LEN(str) DO
	IF PT^ > 96 AND PT^ < 123 THEN PT^ := PT^ - 32; END_IF;
	PT := PT + 1;
END_FOR;
END_FUNCTION

(* POU String/trim, ST *)
FUNCTION trim : STRING
VAR_INPUT
	str : STRING;
END_VAR
VAR
	pos: INT;
END_VAR

(*
version 1.0	6 oct 2006
programmer 	hugo
tested by		tobias

the function deletes all blanks within a string.

*)
trim := str;
REPEAT
	pos := FIND(trim,' ');
	trim := REPLACE(trim,'',1,pos);
UNTIL pos = 0	END_REPEAT;
END_FUNCTION

(* POU String/findB_nonum, ST *)
FUNCTION findB_nonum : INT
VAR_INPUT
	str : STRING;
END_VAR
VAR
	pos: INT;
	pt : POINTER TO BYTE;
END_VAR

(*
version 1.0	6 oct 2006
programmer 	hugo
tested by		tobias

findB_noNum searches str backwards and returns the last position which is not a number.
a number is characterized by a letter "0..9" or "."

*)
pt := ADR(str) + LEN(str) - 1;
findB_nonum := 0;
FOR pos := LEN(str) TO 1 BY -1 DO;
	IF NOT((PT^ > 47 AND PT^ < 58) OR PT^ = 46) THEN
		findB_nonum := pos;
		RETURN;
	END_IF;
	PT := PT - 1;
END_FOR;
END_FUNCTION

(* POU String/findB_Num, ST *)
FUNCTION findB_Num : INT
VAR_INPUT
	str : STRING;
END_VAR
VAR
	pos: INT;
	pt : POINTER TO BYTE;
END_VAR

(*
version 1.0	6 oct 2006
programmer 	hugo
tested by		tobias

findB_Num searches str backward and returns the last position of a number
a number is characterized by a letter "0..9" or "."

*)
pt := ADR(str) + LEN(str) - 1;
findB_Num := 0;
FOR pos := LEN(str) TO 1 BY -1 DO;
	IF (PT^ > 47 AND PT^ < 58) OR PT^ = 46 THEN
		findB_Num := pos;
		RETURN;
	END_IF;
	PT := PT - 1;
END_FOR;
END_FUNCTION

(* POU XTEST/Performance Test/execute_FB, ST *)
FUNCTION_BLOCK execute_FB
VAR_OUTPUT
	ET : REAL;
END_VAR
VAR
	x : fb_list;
	i: DINT;
	start: TIME;
	t: ARRAY[0..150] OF REAL;
	tmax : TIME := t#100ms;
	Y: INT := -1;
	Y_max: INT := 150;
END_VAR

(* this module measures the execution time of all functions in the oscat lib *)
IF Y < Y_max THEN Y := Y+1; ELSE Y := 0; END_IF;
start := TIME();
(* measure the timing overhead *)
i := 0;
REPEAT
	i := i+1;
	x(num := Y, check := TRUE);
UNTIL i > 100000 OR TIME() - start > tmax END_REPEAT;
t[y] := DWORD_TO_REAL(TIME_TO_DWORD(TIME() - start)*1000)/i;

start := TIME();
(* measure the execution time *)
i := 0;
REPEAT
	i := i+1;
	x(num := Y, check := FALSE);
UNTIL i > 100000 OR TIME() - start > tmax END_REPEAT;
t[y] := DWORD_TO_REAL(TIME_TO_DWORD(TIME() - start)*1000)/i - t[y];
t[y] := round(t[y],1);

(* the output is the sum of all modules *)
et := array_sum(ADR(t),SIZEOF(t));
END_FUNCTION_BLOCK

(* POU XTEST/Performance Test/fb_list, ST *)
FUNCTION_BLOCK fb_list
VAR_INPUT
	num : INT;
	check : BOOL;
END_VAR
VAR
	X1: actuator_2P;
	x2 : actuator_3P;
	x3 : actuator_pump;
	x4 : actuator_UD;
	x5 : click;
	x6 : dimm_i;
	x7 : F_Lamp;
	x8 : Pulse_Length;
	x9 : switch_I;
	x10 : Switch_X;
	x11 : timer_1;
	x12 : timer_2;
	x13 : Boiler;
	x14 : Burner;
	x15 : Heat_temp;
	x16 : legionella;
	x17 : temp_ext;
	x18 : FT_Profile;
	x19 : dead_zone2;
	x20 : FT_deriv;
	x21 : FT_IMP;
	x22 : FT_INT;
	x23 : FT_PID;
	x24 : FT_PT1;
	x25 : FT_PT2;
	x26 : FT_TN16;
	x27 : FT_TN64;
	x28 : FT_TN8;
	x29 : hyst_1;
	x30 : hyst_2;
	x31 : Hyst_3;
	x32 : astro;
	x33 : energy;
	x34 : length;
	x35 : pressure;
	x36 : speed;
	x37 : bar_graph;
	x38 : Calibrate;
	x39 : cycle_time;
	x40 : inc_dec;
	x41 : m_d;
	x42 : m_t;
	x43 : m_tx;
	x44 : ontime;
	x45 : gen_rdm;
	x46 : gen_rmp;
	x47 : gen_sin;
	x48 : gen_sqr;
	x49 : pwm_dc;
	x50 : pwm_pw;
	x51 : rmp_B;
	x52 : rmp_soft;
	x53 : rmp_W;
	x54 : delay;
	x55 : delay_4;
	x56 : SH;
	x57 : SH_1;
	x58 : SH_2;
	x59 : SH_T;
	x60 : stair2;
	x61 : FF_D2E;
	x62 : FF_D4E;
	x63 : FF_DRE;
	x64 : FF_JKE;
	x65 : SHR_4E;
	x66 : SHR_4UDE;
	x67 : SHR_8PLE;
	x68 : SHR_8UDE;
	x69 : LTCH;
	x70 : LTCH_4;
	x71 : Byte_to_Bit;
	x72 : DEC_2;
	x73 : DEC_4;
	x74 : DEC_8;
	x75 : B_TRIG;
	x76 : CLK_1ms;
	x77 : CLK_2ms;
	x78 : CLK_4ms;
	x79 : CLK_8ms;
	x80 : clk_div;
	x81 : CLK_Prg;
	x82 : CLK_Pulse;
	x83 : D_Trig;
	x84 : gen_bit;
	x85 : gen_SQ;
	x86 : sequence_4;
	x87 : sequence_8;
	x88 : TP_R;
	x89 : FIFO_16;
	x90 : FIFO_32;
	x91 : STACK_16;
	x92 : STACK_32;
	x93 : matrix;
	x94 : FT_avg;
	x95 : FT_min_max;
	x96 : FT_rmp;
	x97 : ESR_collect;
	x98 : ESR_MON_B8;
	x99 : ESR_MON_R4;
	x100 : ESR_MON_X8;
	x101 : DCF77;
	x102 : holiday;
	x103: Ltime;
	x104 : sun_pos;
	x105 : sun_time;
END_VAR
IF num < 10 THEN
	CASE num OF
	1 : IF check THEN RETURN; ELSE X1; END_IF;
	2 : IF check THEN RETURN; ELSE X2; END_IF;
	3 : IF check THEN RETURN; ELSE X3; END_IF;
	4 : IF check THEN RETURN; ELSE X4; END_IF;
	5 : IF check THEN RETURN; ELSE X5; END_IF;
	6 : IF check THEN RETURN; ELSE X6; END_IF;
	7 : IF check THEN RETURN; ELSE X7; END_IF;
	8 : IF check THEN RETURN; ELSE X8; END_IF;
	9 : IF check THEN RETURN; ELSE X9; END_IF;
	END_CASE;
ELSIF num < 20 THEN
	CASE num OF
	10 : IF check THEN RETURN; ELSE X10; END_IF;
	11 : IF check THEN RETURN; ELSE X11; END_IF;
	12 : IF check THEN RETURN; ELSE X12; END_IF;
	13 : IF check THEN RETURN; ELSE X13; END_IF;
	14 : IF check THEN RETURN; ELSE X14; END_IF;
	15 : IF check THEN RETURN; ELSE X15; END_IF;
	16 : IF check THEN RETURN; ELSE X16; END_IF;
	17 : IF check THEN RETURN; ELSE X17; END_IF;
	18 : IF check THEN RETURN; ELSE X18; END_IF;
	19 : IF check THEN RETURN; ELSE X19; END_IF;
	END_CASE;
ELSIF num < 30 THEN
	CASE num OF
	20 : IF check THEN RETURN; ELSE X20; END_IF;
	21 : IF check THEN RETURN; ELSE X21; END_IF;
	22 : IF check THEN RETURN; ELSE X22; END_IF;
	23 : IF check THEN RETURN; ELSE X23; END_IF;
	24 : IF check THEN RETURN; ELSE X24; END_IF;
	25 : IF check THEN RETURN; ELSE X25; END_IF;
	26 : IF check THEN RETURN; ELSE X26; END_IF;
	27 : IF check THEN RETURN; ELSE X27; END_IF;
	28 : IF check THEN RETURN; ELSE X28; END_IF;
	29 : IF check THEN RETURN; ELSE X29; END_IF;
	END_CASE;
ELSIF num < 40 THEN
	CASE num OF
	30 : IF check THEN RETURN; ELSE X30; END_IF;
	31 : IF check THEN RETURN; ELSE X31; END_IF;
	32 : IF check THEN RETURN; ELSE X32; END_IF;
	33 : IF check THEN RETURN; ELSE X33; END_IF;
	34 : IF check THEN RETURN; ELSE X34; END_IF;
	35 : IF check THEN RETURN; ELSE X35; END_IF;
	36 : IF check THEN RETURN; ELSE X36; END_IF;
	37 : IF check THEN RETURN; ELSE X37; END_IF;
	38 : IF check THEN RETURN; ELSE X38; END_IF;
	39 : IF check THEN RETURN; ELSE X39; END_IF;
	END_CASE;
ELSIF num < 50 THEN
	CASE num OF
	40 : IF check THEN RETURN; ELSE X40; END_IF;
	41 : IF check THEN RETURN; ELSE X41; END_IF;
	42 : IF check THEN RETURN; ELSE X42; END_IF;
	43 : IF check THEN RETURN; ELSE X43; END_IF;
	44 : IF check THEN RETURN; ELSE X44; END_IF;
	45 : IF check THEN RETURN; ELSE X45; END_IF;
	46 : IF check THEN RETURN; ELSE X46; END_IF;
	47 : IF check THEN RETURN; ELSE X47; END_IF;
	48 : IF check THEN RETURN; ELSE X48; END_IF;
	49 : IF check THEN RETURN; ELSE X49; END_IF;
	END_CASE;
ELSIF num < 60 THEN
	CASE num OF
	50 : IF check THEN RETURN; ELSE X50; END_IF;
	51 : IF check THEN RETURN; ELSE X51; END_IF;
	52 : IF check THEN RETURN; ELSE X52; END_IF;
	53 : IF check THEN RETURN; ELSE X53; END_IF;
	54 : IF check THEN RETURN; ELSE X54; END_IF;
	55 : IF check THEN RETURN; ELSE X55; END_IF;
	56 : IF check THEN RETURN; ELSE X56; END_IF;
	57 : IF check THEN RETURN; ELSE X57; END_IF;
	58 : IF check THEN RETURN; ELSE X58; END_IF;
	59 : IF check THEN RETURN; ELSE X59; END_IF;
	END_CASE;
ELSIF num < 70 THEN
	CASE num OF
	60 : IF check THEN RETURN; ELSE X60; END_IF;
	61 : IF check THEN RETURN; ELSE X61; END_IF;
	62 : IF check THEN RETURN; ELSE X62; END_IF;
	63 : IF check THEN RETURN; ELSE X63; END_IF;
	64 : IF check THEN RETURN; ELSE X64; END_IF;
	65 : IF check THEN RETURN; ELSE X65; END_IF;
	66 : IF check THEN RETURN; ELSE X66; END_IF;
	67 : IF check THEN RETURN; ELSE X67; END_IF;
	68 : IF check THEN RETURN; ELSE X68; END_IF;
	69 : IF check THEN RETURN; ELSE X69; END_IF;
	END_CASE;
ELSIF num < 80 THEN
	CASE num OF
	70 : IF check THEN RETURN; ELSE X70; END_IF;
	71 : IF check THEN RETURN; ELSE X71; END_IF;
	72 : IF check THEN RETURN; ELSE X72; END_IF;
	73 : IF check THEN RETURN; ELSE X73; END_IF;
	74 : IF check THEN RETURN; ELSE X74; END_IF;
	75 : IF check THEN RETURN; ELSE X75; END_IF;
	76 : IF check THEN RETURN; ELSE X76; END_IF;
	77 : IF check THEN RETURN; ELSE X77; END_IF;
	78 : IF check THEN RETURN; ELSE X78; END_IF;
	79 : IF check THEN RETURN; ELSE X79; END_IF;
	END_CASE;
ELSIF num < 90 THEN
	CASE num OF
	80 : IF check THEN RETURN; ELSE X80; END_IF;
	81 : IF check THEN RETURN; ELSE X81; END_IF;
	82 : IF check THEN RETURN; ELSE X82; END_IF;
	83 : IF check THEN RETURN; ELSE X83; END_IF;
	84 : IF check THEN RETURN; ELSE X84; END_IF;
	85 : IF check THEN RETURN; ELSE X85; END_IF;
	86 : IF check THEN RETURN; ELSE X86; END_IF;
	87 : IF check THEN RETURN; ELSE X87; END_IF;
	88 : IF check THEN RETURN; ELSE X88; END_IF;
	89 : IF check THEN RETURN; ELSE X89; END_IF;
	END_CASE;
ELSIF num < 100 THEN
	CASE num OF
	90 : IF check THEN RETURN; ELSE X90; END_IF;
	91 : IF check THEN RETURN; ELSE X91; END_IF;
	92 : IF check THEN RETURN; ELSE X92; END_IF;
	93 : IF check THEN RETURN; ELSE X93; END_IF;
	94 : IF check THEN RETURN; ELSE X94; END_IF;
	95 : IF check THEN RETURN; ELSE X95; END_IF;
	96 : IF check THEN RETURN; ELSE X96; END_IF;
	97 : IF check THEN RETURN; ELSE X97; END_IF;
	98 : IF check THEN RETURN; ELSE X98; END_IF;
	99 : IF check THEN RETURN; ELSE X99; END_IF;
	END_CASE;
ELSIF num < 110 THEN
	CASE num OF
	100 : IF check THEN RETURN; ELSE X100; END_IF;
	101 : IF check THEN RETURN; ELSE X101; END_IF;
	102 : IF check THEN RETURN; ELSE X102; END_IF;
	103 : IF check THEN RETURN; ELSE X103; END_IF;
	104 : IF check THEN RETURN; ELSE X104; END_IF;
	105 : IF check THEN RETURN; ELSE X105; END_IF;
	END_CASE;
END_IF;
END_FUNCTION_BLOCK

(* POU Building/electrical/F_Lamp, ST *)
FUNCTION_BLOCK F_Lamp
VAR_INPUT
	SWITCH : BOOL;
	DIMM : BYTE := 255;
	Rst : BOOL;
END_VAR
VAR_OUTPUT
	Lamp : BYTE;
	ontime : REAL;
	cycles : REAL;
	Status : BYTE;
END_VAR
VAR_INPUT CONSTANT
	T_no_Dimm : REAL := 100;
	T_Maintenance : REAL := 15000;
END_VAR
VAR
	runtime : ontime;
	maintenance: BOOL;
END_VAR

(*
version 1.1	8 Feb 2007
programmer 	hugo
tested by		tobias

F_Lamp is an interface to flourescent lamps. its main purpose is to protect flourescent lamps from dimming within the first T_NO_DIMM Time.
If Flourescent Lamps are dimmed during the first 100 hours the lifetime of the lamp is reduced dramatically.
The interface also counts ontime and cycles of the lamp for maintanance purposes.

*)
IF rst THEN
	runtime.rst := TRUE;
	runtime();
	runtime.rst := FALSE;
	ontime := runtime.ontime;
	cycles := runtime.cycles;
	maintenance := FALSE;
ELSE
	runtime(in := Switch);
	ontime := runtime.ontime;
	cycles := runtime.cycles;
END_IF;

IF NOT maintenance AND runtime.ontime >= T_maintenance AND T_Maintenance > 0 THEN
	status := 120;
	maintenance := TRUE;
ELSIF Switch THEN
	IF runtime.ontime < T_no_Dimm THEN
		Lamp := 255;
		STATUS := 111;
	ELSE
		Lamp := DIMM;
		status := 112;
	END_IF;
ELSE
	lamp := 0;
	status := 110;
END_IF;
END_FUNCTION_BLOCK

(* POU Building/electrical/switch_I, ST *)
FUNCTION_BLOCK switch_I
VAR_INPUT
	set : BOOL;
	in : BOOL;
	rst : BOOL;
END_VAR
VAR_INPUT CONSTANT
	T_debounce : TIME := T#10ms;
	T_reconfig : TIME := T#1s;
	T_on_max : TIME := T#0h;
END_VAR
VAR_OUTPUT
	Q : BOOL := 0;
END_VAR
VAR
	state : BYTE := 0;
	edge : BOOL := 0;
	r_edge : BOOL := 0;
	T_on : TIME;
	tx: TIME;
END_VAR

(*
version 1.1	15 sep 2007
programmer 	oscat
tested by		tobias

this is an intelligent switch interface which has an autodetect feature for in and it will detect the type of switch connected automatically
the input can be connected to low active pulses, high active pulses and on/off switch.
it will automatically adjust to the correct type without manual adjustment
a configurable debounce timer will debounce input signals
if t_on_max is set to anything other then 0 the output will be turned off after the max on time is reached.

*)
(* read system time *)
tx := DWORD_TO_TIME(T_PLC_MS());

(* asynchronous set and reset first *)
IF set AND NOT rst THEN
	Q := 1;
	T_on := tx;
ELSIF rst THEN
	Q := 0;
(* check FOR input edge AND start debounce timer *)
ELSIF (in XOR edge) AND NOT (state = 1) THEN
	state := 1;
	T_on := Tx;
(* edge was detected and debounce time elapsed *)
ELSIF (state = 1) AND (Tx - t_debounce >= T_on) THEN
	state := 2;
	(* react on rising or falling edge depending on r_edge *)
	IF r_edge XOR in THEN Q := NOT Q; END_IF;
(* wait for T_reconfig and adjust r_edge *)
ELSIF state = 2 AND Tx - t_reconfig >= T_on THEN
	r_edge := in;
END_IF;
IF Q AND T_on_max > t#0ms AND Tx >= T_on + T_on_max THEN
	Q := FALSE;
END_IF;
edge := in;

(* revision history

hm	4 aug 2006	rev 1.0
	original version

hm	15.9.2007	rev 1.1
	replaced Time() with T_PLC_MS for compatibility and performance reasons

*)
END_FUNCTION_BLOCK

(* POU Building/electrical/Switch_X, ST *)
FUNCTION_BLOCK Switch_X
VAR_INPUT
	IN1 : BOOL;
	IN2 : BOOL;
	IN3 : BOOL;
	IN4 : BOOL;
	IN5 : BOOL;
	IN6 : BOOL;
END_VAR
VAR_OUTPUT
	Q1 : BOOL;
	Q2 : BOOL;
	Q3 : BOOL;
	Q4 : BOOL;
	Q5 : BOOL;
	Q6 : BOOL;
	Q31 : BOOL;
	Q41 : BOOL;
	Q51 : BOOL;
	Q61 : BOOL;
	Q32 : BOOL;
	Q42 : BOOL;
	Q52 : BOOL;
	Q62 : BOOL;
END_VAR
VAR_INPUT CONSTANT
	t_debounce : TIME := t#50ms;
END_VAR
VAR
	init : BOOL;
	T1, T2, T3, T4, T5, T6 : TOF;
	tx: TIME;
	x1: BOOL;
	x2: BOOL;
	E1, E2 : BOOL;
END_VAR

(*
version 1.0	15 Feb 2007
programmer 	oscat
tested by		tobias

*)
(* initialize on startup *)
IF NOT init THEN
	init := TRUE;
	IF t_debounce < t#50ms THEN tx := t#50ms; ELSE tx := t_debounce; END_IF;
	T1(PT := Tx);
	T2(PT := Tx);
	T3(PT := Tx);
	T4(PT := Tx);
	T5(PT := Tx);
	T6(PT := Tx);
ELSE
	Q1 := FALSE;
	Q2 := FALSE;
	Q3 := FALSE;
	Q4 := FALSE;
	Q5 := FALSE;
	Q6 := FALSE;
	Q31 := FALSE;
	Q41 := FALSE;
	Q51 := FALSE;
	Q61 := FALSE;
	Q32 := FALSE;
	Q42 := FALSE;
	Q52 := FALSE;
	Q62 := FALSE;
END_IF;

(* read inputs and debounce *)
	T1(IN := IN1);
	T2(IN := IN2);
	T3(IN := IN3);
	T4(IN := IN4);
	T5(IN := IN5);
	T6(IN := IN6);

(* detect edge of IN1 and IN2 *)
IF t1.Q AND NOT E1 THEN X1 := TRUE; END_IF;
IF t2.Q AND NOT E2 THEN X2 := TRUE; END_IF;

IF t1.Q THEN
	IF t3.q THEN
		q31 := TRUE;
		X1 := FALSE;
	ELSIF t4.q THEN
		q41 := TRUE;
		X1 := FALSE;
	ELSIF t5.q THEN
		q51 := TRUE;
		X1 := FALSE;
	ELSIF t6.q THEN
		q61 := TRUE;
		X1 := FALSE;
	END_IF;
ELSIF t2.Q THEN
	IF t3.q THEN
		q32 := TRUE;
		X2 := FALSE;
	ELSIF t4.q THEN
		q42 := TRUE;
		X2 := FALSE;
	ELSIF t5.q THEN
		q52 := TRUE;
		X2 := FALSE;
	ELSIF t6.q THEN
		q62 := TRUE;
		X2 := FALSE;
	END_IF;
(* in1 was active alone *)
ELSIF NOT T1.Q AND E1 AND X1 THEN
	Q1 := TRUE;
	X1 := FALSE;
ELSIF NOT T2.Q AND E2 AND X2 THEN
	Q2 := TRUE;
	X2 := FALSE;
ELSIF T3.Q THEN
	Q3 := TRUE;
ELSIF T4.Q THEN
	Q4 := TRUE;
ELSIF T5.Q THEN
	Q5 := TRUE;
ELSIF T6.Q THEN
	Q6 := TRUE;
END_IF;

(* save state of in1 and in2 *)
E1 := T1.Q;
E2 := T2.Q;
END_FUNCTION_BLOCK

(* POU Building/electrical/timer_1, ST *)
FUNCTION_BLOCK timer_1
VAR_INPUT
	DT_in : DT;
	start_time : TOD;
	duration : TIME;
	start_day : INT := 0;
END_VAR
VAR_OUTPUT
	Q : BOOL;
END_VAR
VAR
	last_check : TIME := T#0s;
	last: DATE := D#2041-01-01;
	dat: DATE;
	init : BOOL;
	tx: TIME;
	pulse_start: TIME;
END_VAR

(*
version 1.5	1. okt 2007
programmer 	oscat
tested by		tobias

this is a simple timer that generates an output pulse once a day if start_day = 0.
if start_day is a number from 1 .. 7 then a output pulse is generated for the respective weekday 1 = monday.
the output pulse width can be programmed, if set to 0 a pulse is generated for one cycle only.

*)
(* read system timer *)
tx := DWORD_TO_TIME(T_PLC_MS());

(* init on startup *)
IF NOT init THEN
	init := TRUE;
	last_check := tx - t#100ms;
END_IF;

(* check every 100ms *)
IF tx - last_check >= T#100ms THEN
	dat := DT_TO_DATE(dt_in);
	IF NOT Q AND (start_day = 0 OR start_day = weekday(dat)) AND dat <> last AND DT_TO_TOD(dt_in) >= start_time THEN
		Q := TRUE;
		last := dat;
		pulse_start := tx;
	ELSIF Q AND tx - pulse_start >= duration THEN
		Q := FALSE;
	END_IF;
	last_check := tx;
END_IF;

(*
1.12.2006 hm		rev 1.1
	corrected an error with pulse width = 0.

25.12.2006 hm	rev 1.2
	corrected an error when timer overflows.

14.apr 2007 hm	rev 1.3
	corrected an error while while output would not go active when start year would be 1970.
	increase accuracy by checking every 100ms
	added init section to compensate for timer overflow

15.9.2007	hm		rev 1.4
	replaced Time() with T_PLC_MS for compatibility and performance reasons

hm	1. okt 2007		rev 1.5
	corrected an error while output would not stay active over midnight.

*)
END_FUNCTION_BLOCK

(* POU Building/HLK/Heat_temp, ST *)
FUNCTION_BLOCK Heat_temp
VAR_INPUT
	T_ext : REAL;
	Offset : REAL;
	t_req : REAL;
END_VAR
VAR_INPUT CONSTANT
	TY_max : REAL := 70;
	TY_min : REAL := 20;
	T_int : REAL := 20;
	TY_config : REAL := 50;
	T_ext_config : REAL := -15;
	C : REAL := 1.33;
END_VAR
VAR_OUTPUT
	Ty : REAL;
END_VAR
VAR
END_VAR

(*
version 1.0	27 jan 2007
programmer 	hugo
tested by		tobias

Heat_Temp calculates a heat characteristic based on the formula: tv=ti+(tvmax-ti)*((ti-tau)/(ti-taumin))^(1/n)
while
tv necessary heating temperature.
ti internal room temperature (20°C)
tau current external temperature
external temperature to determine characteristics
C exponent for heating system (normally 1,33 or 1,1 for floor heating)

The two additional inputs TY_min and TY_max set limits for the output TY, while an offset inputs allows to rise or lower the room temperature.

*)
IF t_ext > t_int + Offset THEN
	ty := t_int + offset;
ELSE
Ty := T_int - offset + (TY_config - T_int) * EXPT((T_int - offset - T_ext) / (T_int - offset - T_ext_config),1 / C);
END_IF;
IF t_req > ty THEN ty := t_req; END_IF;
ty := LIMIT(TY_min, ty, TY_max);



(*

tv=ti+(tvmax-ti)*((ti-tau)/(ti-taumin))^(1/n)

tv aktuelle Vorlauftemp.
ti Raumtemperatur innen (20°C)
tau aktuelle Außentemperatur
taumin minimale Außentemperatur -12°C oder -15°C
n Heizkörperexponent (meistens 1,33)
Fußbodenheizung = 1,1
Wandheizung 1,3

Normen z. B. DIN 4703, DIN 4725 oder die Literatur, z. B Recknagel Abschnitt 1.3.5.

*)
END_FUNCTION_BLOCK

(* POU Building/HLK/legionella, ST *)
FUNCTION_BLOCK legionella
VAR_INPUT
	manual : BOOL;
	temp_boiler : REAL;
	temp_return : REAL := 100;
	DT_in: DT;
	rst : BOOL;
END_VAR
VAR_INPUT CONSTANT
	T_start: TOD := tod#03:00:00;
	day : INT := 7;
	temp_set : REAL := 70;
	temp_offset : REAL := 10;
	temp_hys : REAL := 5;
	t_max_heat: TIME := t#10m;
	t_max_ret : TIME := t#10m;
	tp_0: TIME := t#5m;
	tp_1: TIME := t#5m;
	tp_2: TIME := t#5m;
	tp_3: TIME := t#5m;
	tp_4: TIME := t#5m;
	tp_5: TIME := t#5m;
	tp_6: TIME := t#5m;
	tp_7: TIME := t#5m;
END_VAR
VAR_OUTPUT
	Heat : BOOL;
	pump : BOOL;
	valve0 : BOOL;
	valve1 : BOOL;
	valve2 : BOOL;
	valve3 : BOOL;
	valve4 : BOOL;
	valve5 : BOOL;
	valve6 : BOOL;
	valve7 : BOOL;
	run: BOOL;
	Status : BYTE;
END_VAR
VAR
	X1: timer_1;
	x2: sequence_8;
	x3: hyst_1;
	init: BOOL;
END_VAR

(*
version 1.1	17. jan 2007
programmer 	oscat
tested by		hans

Legionella is a complete sequencer for up to 8 hot water lines that need to be sterilzed periodically.
legionella needs a DT input with the appropriate time, usually gererated by the rtc of the system. for system independence this time is connected externally.
T_start is the time when sterilazation should be started and day is the day_of_week when it should be performed (1=Monday and 7=sunday).
so sterilazation is autioimatically performed once a week at a specified time.
temp_set and temp_hys and temp_offset specify the boiler temperatur nedded for sterilization. as a defaut Temp_set is set to 70 deg C and Temp_hys is set to 5 deg C and temp_offset is 10 deg C.
a temp boiler input reads the boiler temperature of the hot water tank.
after a start pulse is gererated by the weekly timer or a manual test input the sequence is started:
1. the boiler is heated to temp_set + temp_offset + temp_hys = 85 deg C unless chaged at setup.
	the heat output is turned on and tells the heater to turn heating on. if the temp is not reached for a time of t_max_heat (10 min) the error output is set and the sequence is stopped.
2. after the specified temperature is reached, the output valve0 and pump is turned on and starts sterilization of line0 until temp_return has reached temp_set and continues to sterilize for a time of tp_0 (5 min default).
	if tmep_set is not reached at the temp_return_input then the error output is set and the sequence will be stopped.
	if there is no temp sensor for temp_return (the temperature at the return point for the circulation pump pls set this imput to a value greater then temp_set (by default use 100 deg C).
	in this case sterilization is performed for the default times without monitoring the return temp.
3. this sequence is repeated for up to valves.

connection scheme:

temp_boiler:	input oif the boiler temperature sensor.
temp_hys:		config value for the heater hysteresis, preset to 5 deg C.
temp_offset:	config value for the heater temp_offset against temp_set, preset to 10 deg C.
temp_set:		config value for the specified sterilization temperature, preset to 70 deg C.
temp_return:	input of the circulation return line temperature sensor, if not availabe set this value to 100 deg C.
manual:		manual input to start the sterilization by hand for diagnostic purposes, rising edge active, leave low for automatic operation.
DT_in:			date,time input supplied by a external real time clock.
T_start:		time of day when the sterilization should be started.
day:			config value for day of week when the process should be started, preset to sunday.
t_max_hest:	tmax time to be needed for the heater to heat the hot water tank to the specified value, preset to 10 min.

*)
(* startup initialization *)
IF NOT init THEN
	init := TRUE;
	X1.start_day := day;
	X1.start_time := T_start;
	X3.low := Temp_offset + temp_set;
	X3.high := Temp_hys + X3.low;
	X2.wait0 := T_max_heat;
	X2.delay0 := TP_0;
	X2.delay1 := TP_1;
	X2.delay2 := TP_2;
	X2.delay3 := TP_3;
	X2.delay4 := TP_4;
	X2.delay5 := TP_5;
	X2.delay6 := TP_6;
	X2.delay7 := TP_7;
	X2.wait1 := T_max_ret;
	X2.wait2 := T_max_ret;
	X2.wait3 := T_max_ret;
	X2.wait4 := T_max_ret;
	X2.wait5 := T_max_ret;
	X2.wait6 := T_max_ret;
	X2.wait7 := T_max_ret;
	X2();
END_IF;

(* oerational code *)
X1(DT_in := DT_in);
IF X1.Q OR manual OR x2.run THEN
	X3(in := temp_boiler);
	X2.in0 := X3.Q OR x3.win;
	X2.in1 := temp_return >= temp_set;
	X2.in2 := x2.in1;
	X2.in3 := x2.in1;
	X2.in4 := x2.in1;
	X2.in5 := x2.in1;
	X2.in6 := x2.in1;
	X2.in7 := x2.in1;
	X2.rst := rst;
	X2(start := X1.Q OR manual);
	run := x2.run;
	pump := x2.any;
	Heat := NOT X3.Q AND x2.run;
	valve0 := X2.Q0;
	valve1 := X2.Q1;
	valve2 := X2.Q2;
	valve3 := X2.Q3;
	valve4 := X2.Q4;
	valve5 := X2.Q5;
	valve6 := X2.Q6;
	valve7 := X2.Q7;
	pump := X2.any;
	status := X2.status;
ELSE;
	X2(start :=0);
	status := x2.status;
END_IF;

(* revision history

hm 17.jan 2007	rev 1.1
	rewritten to st for higher performance
	changes eeror output to esr compatible status output
*)
END_FUNCTION_BLOCK

(* POU Logic/generators/sequence_8, ST *)
FUNCTION_BLOCK sequence_8
VAR_INPUT
	in0 : BOOL := TRUE;
	in1 : BOOL := TRUE;
	in2 : BOOL := TRUE;
	in3 : BOOL := TRUE;
	in4 : BOOL := TRUE;
	in5 : BOOL := TRUE;
	in6 : BOOL := TRUE;
	in7 : BOOL := TRUE;
	start : BOOL;
	rst : BOOL;
	wait0 : TIME := t#0s;
	delay0 : TIME := t#0s;
	wait1 : TIME := t#0s;
	delay1 : TIME := t#0s;
	wait2 : TIME := t#0s;
	delay2 : TIME := t#0s;
	wait3 : TIME := t#0s;
	delay3 : TIME := t#0s;
	wait4 : TIME := t#0s;
	delay4 : TIME := t#0s;
	wait5 : TIME := t#0s;
	delay5 : TIME := t#0s;
	wait6 : TIME := t#0s;
	delay6 : TIME := t#0s;
	wait7 : TIME := t#0s;
	delay7 : TIME := t#0s;
END_VAR
VAR_INPUT CONSTANT
	stop_on_error : BOOL := FALSE;
END_VAR
VAR_OUTPUT
	Q0 : BOOL;
	Q1 : BOOL;
	Q2 : BOOL;
	Q3 : BOOL;
	Q4 : BOOL;
	Q5 : BOOL;
	Q6 : BOOL;
	Q7 : BOOL;
	any : BOOL;
	run: BOOL;
	step : INT := -1;
	status : BYTE;
END_VAR
VAR
	last : TIME;
	edge : BOOL;
	tx: TIME;
	init: BOOL;
END_VAR

(*
version 1.4	17 sep 2007
programmer 	oscat
tested by		hans

sequence_8 enables run when a low to high transition is present on start.
a low to high transition on start will restart the sequencer at any time while a rst will hold the sequencer in reset while true.
after run is enabled with a rising edge on start the sequencer waits for wait0 on in0 to enable q0 which stays on for delay0.
the next cycle starts with wait1, continues with delay 1 and so on...
if an edge is not detected during the wait period, the sequencer will then display the error number on the status output.
The status numbers are 1 .. 8 for erros in step 0..7.
after the last step that sets q7, the sequencer leaves q7 on for delay7 and then resets to the initial state.
a step output will indicate the current step of the sequencer and will also be present with a fault condition.
after the first output is turened on the sequencer switches from q0 to q1 and so on, at any time there is only one output enabled.
if an input signal is not detected during a wait period, the sequencer will display the error number ( 1 for in0, 2 for in1 .... ).
when an error is present and the config variable stop_on_error is set then the sequencer will stop. otherwise it will continue.
The status output will also display 110 for waiting and 111 sequece running.

*)
(* read sps timer *)
tx := DWORD_TO_TIME(T_PLC_MS());

(* initialize on startup *)
IF NOT init THEN
	last := tx;
	init := TRUE;
	status := 110;
END_IF;

(* asynchronous reset *)
IF rst THEN
	step := -1;
	Q0 := 0;
	Q1 := 0;
	Q2 := 0;
	Q3 := 0;
	Q4 := 0;
	Q5 := 0;
	Q6 := 0;
	Q7 := 0;
	status := 110;
	run := 0;

(* edge on start input restarts the sequencer *)
ELSIF start AND NOT edge THEN
	step := 0;
	last := tx;
	status := 111;
	Q0 := 0;
	Q1 := 0;
	Q2 := 0;
	Q3 := 0;
	Q4 := 0;
	Q5 := 0;
	Q6 := 0;
	Q7 := 0;
	run := 1;
END_IF;
edge := start;

(* check if stop on error is necessary *)
IF status > 0 AND status < 100 AND stop_on_error THEN RETURN; END_IF;

(* sequence is running *)
IF run AND step = 0 THEN
	IF NOT q0 AND in0 AND tx - last <= wait0 THEN
		Q0 := TRUE;
		last := tx;
	ELSIF NOT q0 AND tx - last > wait0 THEN
		status := 1;
		run := FALSE;
	ELSIF q0 AND tx - last >= delay0 THEN
		step := 1;
		last := tx;
	END_IF;
END_IF;
IF run AND step = 1 THEN
	IF NOT q1 AND in1 AND tx - last <= wait1 THEN
		Q0 := FALSE;
		Q1 := TRUE;
		last := tx;
	ELSIF NOT q1 AND Tx - last > wait1 THEN
		status := 2;
		q0 := FALSE;
		run := FALSE;
	ELSIF q1 AND tx - last >= delay1 THEN
		step := 2;
		last := tx;
	END_IF;
END_IF;
IF run AND step = 2 THEN
	IF NOT q2 AND in2 AND tx - last <= wait2 THEN
		Q1 := FALSE;
		Q2 := TRUE;
		last := tx;
	ELSIF NOT q2 AND Tx - last > wait2 THEN
		status := 3;
		q1 := FALSE;
		run := FALSE;
	ELSIF q2 AND tx - last >= delay2 THEN
		step := 3;
		last := tx;
	END_IF;
END_IF;
IF run AND step = 3 THEN
	IF NOT q3 AND in3 AND tx - last <= wait3 THEN
		Q2 := FALSE;
		Q3 := TRUE;
		last := tx;
	ELSIF NOT q3 AND Tx - last > wait3 THEN
		status := 4;
		q2 := FALSE;
		run := FALSE;
	ELSIF q3 AND tx - last >= delay3 THEN
		step := 4;
		last := tx;
	END_IF;
END_IF;
IF run AND step = 4 THEN
	IF NOT q4 AND in4 AND tx - last <= wait4 THEN
		Q3 := FALSE;
		Q4 := TRUE;
		last := tx;
	ELSIF NOT q4 AND Tx - last > wait4 THEN
		status := 5;
		q3 := FALSE;
		run := FALSE;
	ELSIF q4 AND tx - last >= delay4 THEN
		step := 5;
		last := tx;
	END_IF;
END_IF;
IF run AND step = 5 THEN
	IF NOT q5 AND in5 AND tx - last <= wait5 THEN
		Q4 := FALSE;
		Q5 := TRUE;
		last := tx;
	ELSIF NOT q5 AND Tx - last > wait5 THEN
		status := 6;
		q4 := FALSE;
		run := FALSE;
	ELSIF q5 AND tx - last >= delay5 THEN
		step := 6;
		last := tx;
	END_IF;
END_IF;
IF run AND step = 6 THEN
	IF NOT q6 AND in6 AND tx - last <= wait6 THEN
		Q5 := FALSE;
		Q6 := TRUE;
		last := tx;
	ELSIF NOT q6 AND Tx - last > wait6 THEN
		status := 7;
		q5 := FALSE;
		run := FALSE;
	ELSIF q6 AND tx - last >= delay6 THEN
		step := 7;
		last := tx;
	END_IF;
END_IF;
IF run AND step = 7 THEN
	IF NOT q7 AND in7 AND tx - last <= wait7 THEN
		Q6 := FALSE;
		Q7 := TRUE;
		last := tx;
	ELSIF NOT q7 AND Tx - last > wait7 THEN
		status := 8;
		q6 := FALSE;
		run := FALSE;
	ELSIF q7 AND tx - last >= delay7 THEN
		step := -1;
		Q7 := FALSE;
		Run := FALSE;
		status := 110;
	END_IF;
END_IF;
any := q0 OR q1 OR q2 OR q3 OR q4 OR q5 OR q6 OR q7;

(*
hm 1.10.06		rev 1.1
	corrected delay logic to be after event and not before
	added any output

hm 1.12.06		rev 1.2
	corrected failure in sequence logic.
	added init at startup to prevent from initial statuss after start.

hm 17.1.2007		rev 1.3
	changed output fault to status for better compatibility with other modules (ESR)
	added stop on error functionality and setup variable
	default for inputs in0..7 is true.
	renames variable state to step

hm	17.sep 2007		rev 1.4
	replaced time() with T_PLC_MS() for compatibility reasons

*)
END_FUNCTION_BLOCK

(* POU engineering/control/hyst_1, ST *)
FUNCTION_BLOCK hyst_1
VAR_INPUT
	In : REAL;
	high : REAL;
	low : REAL;
END_VAR
VAR_OUTPUT
	Q : BOOL := 0;
	win : BOOL := 0;
END_VAR
VAR
END_VAR

(*
	version 1.0	4 aug 2006
	programmer 	hugo
	tested BY		tobias

this hysteresis function switches the output high if the input signal reaches obove high and will switch to low when the input falls back below low value.
a separate output mid is set if the input stays between low and high value.

*)
IF Q THEN
	IF in < low THEN q := FALSE; END_IF;
ELSE
	IF in > high THEN q := TRUE; END_IF;
END_IF;
win := in > low AND in < high;
END_FUNCTION_BLOCK

(* POU Building/HLK/temp_ext, ST *)
FUNCTION_BLOCK temp_ext
VAR_INPUT
	t_ext1 : REAL;
	t_ext2 : REAL;
	t_ext3 : REAL;
	t_ext_config : BYTE := 0;
	dt_in : DT;
END_VAR
VAR_INPUT CONSTANT
	t_ext_min : REAL := -40;
	t_ext_max : REAL := 60;
	t_ext_default : REAL := -10;
	heat_period_start : DATE := D#1970-9-1;
	heat_period_stop : DATE := D#1970-4-30;
	cool_period_start : DATE := D#1970-4-1;
	cool_period_stop : DATE := D#1970-9-30;
	heat_start_temp_day : REAL := 15;
	heat_start_temp_night : REAL := 10;
	heat_stop_temp : REAL := 18;
	cool_start_temp_day : REAL := 26;
	cool_start_temp_night : REAL := 26;
	cool_stop_temp : REAL := 24;
	start_day : TOD := tod#09:00;
	start_night : TOD := tod#21:00;
	cycle_time : TIME := t#10m;
END_VAR
VAR_OUTPUT
	t_ext : REAL;
	heat : BOOL;
	cool : BOOL;
END_VAR
VAR
	tx: TIME;
	last_run: TIME;
	init: BOOL;
	cool_start: DATE;
	cool_stop: DATE;
	heat_start: DATE;
	heat_stop: DATE;
	xdate: DATE;
	day: BOOL;
END_VAR


(*
version 1.1	15 sep 2007
programmer 	hugo
tested by		tobias

temp_ext measures and processes ext temperature and decides if heating or cooling is needed.

 the measurement of t_ext has 3 inputs which can be configured in different ways:
	t_ext_config = 0 means the ext temp is the avg of the 3 external temperatures, this mode is the default mode.
	t_ext_config = 1 means t_ext1 is used.
	t_ext_config = 2 means t_ext1 is used.
	t_ext_config = 3 means t_ext1 is used.
	t_ext_config = 4 means t_ext_default is used.
	t_ext_config = 5 means the lowest of the 3 external temperatures is used.
	t_ext_config = 6 means the higest externnal temperature is used.
	t_ext_config = 7 means the midlle external temperature is used, if there are only two working, the lowest is used.
	in any config mode, an external temperature higher then t_ext_max or lower then t_ext_min is ignored to prevent from temperatures caused by broken sensors or wires.
	if no external temperature is available, a default value (t_ext_default) is used.
	if you have only one external sensor, connect the 3 inputs to the same sensor, or select the right input with t_ext_config.

heating or cooling is enabled during heating / cooling period when the day or night start temperature is reached for at least the specified delay time and will be disabled after the stop temperature is reached. 
t_ext output can be used by other modules to determine the correct system temperature for heating or cooling.

*)
IF NOT init THEN
	init := TRUE;
	heat_start := set_Date(1972,month(heat_period_start),day_of_month(heat_period_start));
	heat_stop := set_Date(1972,month(heat_period_stop),day_of_month(heat_period_stop));
	cool_start := set_Date(1972,month(cool_period_start),day_of_month(cool_period_start));
	cool_stop := set_Date(1972,month(cool_period_stop),day_of_month(cool_period_stop));
END_IF;

(* read system time *)
tx := DWORD_TO_TIME(T_PLC_MS());

(* for efficiency exit isf this program has been executed less then 1min ago *)
IF tx - last_run < cycle_time THEN RETURN; END_IF;

(* calculate frequently used variables *)
xdate := set_Date(1972,month(DT_TO_DATE(dt_in)),day_of_month(DT_TO_DATE(dt_in)));
day := DT_TO_TOD(dt_in) >= start_day AND  DT_TO_TOD(dt_in) < start_night;

(* read the correct external temperature depending on the t_ext_config setting *)
t_ext := multi_in(t_ext1, t_ext2, t_ext3, t_ext_default, t_ext_min, t_ext_max, t_ext_config);

(* dtermine heating *)
IF (heat_start <= heat_stop AND xdate >= heat_start AND xdate <= heat_stop) OR (heat_start > heat_stop AND (xdate >= heat_start OR xdate <= heat_stop)) THEN
	(* heating period id true check for temperature *)
	IF day AND t_ext <= heat_start_temp_day THEN
		heat := TRUE;
	ELSIF NOT day AND t_ext <= heat_start_temp_night THEN
		heat := TRUE;
	ELSIF t_ext >= heat_stop_temp THEN
		heat := FALSE;
	END_IF;
ELSE
	heat := FALSE;
END_IF;

(* dtermine cooling *)
IF (cool_start <= cool_stop AND xdate >= cool_start AND xdate <= cool_stop) OR (cool_start > cool_stop AND (xdate >= cool_start OR xdate <= cool_stop)) THEN
	(* cooling period is true check for temperature *)
	IF day AND t_ext >= cool_start_temp_day THEN
		cool := TRUE;
	ELSIF NOT day AND t_ext >= cool_start_temp_night THEN
		cool := TRUE;
	ELSIF t_ext <= cool_stop_temp THEN
		cool := FALSE;
	END_IF;
ELSE
	cool := FALSE;
END_IF;

last_run := tx;

(* revision history
hm	6 dec 2006		rev 1.0
	original version

hm	15.9.2007		rev 1.1
	replaced Time() with T_PLC_MS for compatibility and performance reasons

*)
END_FUNCTION_BLOCK

(* POU engineering/sensor/multi_in, ST *)
FUNCTION multi_in : REAL
VAR_INPUT
	in_1 : REAL;
	in_2 : REAL;
	in_3 : REAL;
	default : REAL;
	in_min : REAL;
	in_max : REAL;
	mode : BYTE;
END_VAR
VAR
	count: INT;
	F1: BOOL;
	F2: BOOL;
	F3: BOOL;
END_VAR

(*

version 1.1	1 jan 2007
programmer 	oscat
tested by		hugo

multi_in is a signal conditioning function ehich can be configured in 8 different ways.
it is used to read multiple sensors for the same value and protect the user from broken sensors or invalid data from sensors.

multi_in can be configured in different ways:
	mode = 0 means the the avg of the 3 inputs is used, this mode is the default mode.
	mode = 1 means in_1 is used.
	mode = 2 means in_2 is used.
	mode = 3 means in_3 is used.
	mode = 4 means default is used.
	mode = 5 means the lowest of the 3 external temperatures is used.
	mode = 6 means the higest externnal temperature is used.
	mode = 7 means the midlle input is used, if there are only two working, the lowest input is used.
	mode > 7 ,eans output is 0 at all times.
	in any config mode, an input higher then in_max or lower then in_min is ignored to prevent values from broken sensors or wires.
	if all inputs are higher then in_max or lower then in_min, a default value (default) is used.
*)
IF  in_1 > in_min AND in_1 < in_max THEN F1 := TRUE; ELSE F1 := FALSE; END_IF;
IF  in_2 > in_min AND in_2 < in_max THEN F2 := TRUE; ELSE F2 := FALSE; END_IF;
IF  in_2 > in_min AND in_3 < in_max THEN F3 := TRUE; ELSE F3 := FALSE; END_IF;

CASE mode OF
0:	count := 0;
	IF F1 THEN
		count := count + 1;
		multi_in := in_1;
	ELSE
		multi_in := 0;
	END_IF;
	IF F2 THEN
		count := count + 1;
		multi_in := multi_in + in_2;
	END_IF;
	IF F3 THEN
		count := count + 1;
		multi_in := multi_in + in_3;
	END_IF;
	IF count = 0 THEN
		multi_in := default;
	ELSE
		multi_in := multi_in / count;
	END_IF;

1:	IF F1 THEN multi_in := in_1; ELSE multi_in := default; END_IF;

2:	IF F2 THEN multi_in := in_2; ELSE multi_in := default; END_IF;

3:	IF F3 THEN multi_in := in_3; ELSE multi_in := default; END_IF;

4:	multi_in := default;

5:	IF F1 THEN multi_in := in_1; ELSE multi_in := in_max; END_IF;
	IF F2 AND in_2 < multi_in THEN multi_in := in_2; END_IF;
	IF F3 AND in_3 < multi_in THEN multi_in := in_3; END_IF;
	IF multi_in = in_max THEN multi_in := default; END_IF;

6:	IF F1 THEN multi_in := in_1; ELSE multi_in := in_min; END_IF;
	IF F2 AND in_2 > multi_in THEN multi_in := in_2; END_IF;
	IF F3 AND in_3 > multi_in THEN multi_in := in_3; END_IF;
	IF multi_in = in_min THEN multi_in := default; END_IF;

7:	IF F1 AND F2 AND F3 THEN multi_in := mid3(in_1, in_2, in_3);
	ELSIF F1 AND F2 THEN multi_in := MIN(in_1, in_2);
	ELSIF F1 AND F3 THEN multi_in := MIN(in_1, in_3);
	ELSIF F2 AND F3 THEN multi_in := MIN(in_2, in_3);
	ELSIF F1 THEN multi_in := in_1;
	ELSIF F2 THEN multi_in := in_2;
	ELSIF F3 THEN multi_in := in_3;
	ELSE multi_in := default;
	END_IF;

END_CASE;

(*
hm 1.1.2007	rev 1.1
	changed midr to mid3 function

*)
END_FUNCTION

(* POU mathematical/mid3, ST *)
FUNCTION mid3 : REAL
VAR_INPUT
	in1 : REAL;
	in2 : REAL;
	in3 : REAL;
END_VAR
VAR
END_VAR

(*
version 1.1	1 jan 2007
programmer 	hugo
tested by		tobias

returns the mid value of 3 real inputs.

*)
IF (in1 <= in2) AND (in1 >= in3) OR (in1 >= in2) AND (in1 <= in3) THEN
	mid3 := in1;
ELSIF (in2 <= in1) AND (in2 >= in3) OR (in2 >= in1) AND (in2 <= in3) THEN
	mid3 := in2;
ELSE
	mid3 := in3;
END_IF;

(*
hm	1.1.2007	rev 1.1
	rewrote the function for better performance

*)
END_FUNCTION

(* POU engineering/automation/FT_Profile, ST *)
FUNCTION_BLOCK FT_Profile
VAR_INPUT
	K : REAL := 1;
	O : REAL := 0;
	M : REAL := 1;
	E : BOOL;
END_VAR
VAR_INPUT CONSTANT
	value_0 : REAL;
	time_1 : TIME;
	value_1 : REAL;
	time_2 : TIME;
	value_2 : REAL;
	time_3 : TIME;
	value_3 : REAL;
	time_10 : TIME;
	value_10 : REAL;
	time_11 : TIME;
	value_11 : REAL;
	time_12 : TIME;
	value_12 : REAL;
	time_13 : TIME;
	value_13 : REAL;
END_VAR
VAR_OUTPUT
	Y : REAL;
	RUN : BOOL;
	ET : TIME;
END_VAR
VAR
	tx : TIME;
	edge : BOOL;
	state: BYTE;
	ta: TIME;
	tb: TIME;
	t0 : TIME;
	temp: REAL;
	va: REAL;
	vb: REAL;
END_VAR

(*
version 1.1	15 sep 2007
programmer 	tobias
tested by		hugo

FT_Profile generates an output signal which is defined by values over a time scale.
the different values are connected by ramps between the individual values.
a rising edge on E starts the output signal generation and E = True can delay time_3 / value_3 as long as it stays true.
an additional multiplier K can be used to multiply the output and an offset O can be added to the output dynamically.
*)
(* read system time *)
tx := DWORD_TO_TIME(T_PLC_MS());

(* determine start condition *)
IF E AND NOT edge THEN
	RUN := TRUE;
	ET := t#0s;
	t0 := tx;
	ta := tx;
	tb := multime(time_1, M);
	va := value_0;
	vb := value_1;
	temp := value_0;
	state := 1;
END_IF;
edge := E;

(* generate startup profile *)
IF run THEN
	CASE state OF
		1:	IF tx - ta >= tb THEN
				ta := ta + tb;
				tb := multime(time_2 - time_1, M);
				va := value_1;
				vb := value_2;
				temp := value_1;
				state := 2;
			ELSE
				temp := ((vb - va) * TIME_TO_REAL(tx - ta) / TIME_TO_REAL(tb) + va);
			END_IF;
		2:	IF tx - ta >= tb THEN
				ta := ta + tb;
				tb := multime(time_3 - time_2, M);
				va := value_2;
				vb := value_3;
				temp := value_2;
				state := 3;
			ELSE
				temp := ((vb - va) * TIME_TO_REAL(tx - ta) / TIME_TO_REAL(tb) + va);
			END_IF;
		3:	IF tx - ta >= tb THEN
				ta := ta + tb;
				tb := multime(time_10 - time_3, M);
				va := value_3;
				vb := value_10;
				temp := value_3;
				state := 4;
			ELSE
				temp := ((vb - va) * TIME_TO_REAL(tx - ta) / TIME_TO_REAL(tb) + va);
			END_IF;
		4 :	IF tx - ta >= tb THEN
				ta := ta + tb;
				tb := multime(time_11 - time_10, M);
				va := value_10;
				vb := value_11;
				temp := value_10;
				IF E THEN state := 5; ELSE state := 6; END_IF;
			ELSE
				temp := ((vb - va) * TIME_TO_REAL(tx - ta) / TIME_TO_REAL(tb) + va);
			END_IF;
		5:	(* extend the signal while E is true *)
			IF E THEN
				ta := tx;
			ELSE
				state := 6;
			END_IF;
		6:	IF tx - ta >= tb THEN
				ta := ta + tb;
				tb := multime(time_12 - time_11, M);
				va := value_11;
				vb := value_12;
				temp := value_11;
				state := 7;
			ELSE
				temp := ((vb - va) * TIME_TO_REAL(tx - ta) / TIME_TO_REAL(tb) + va);
			END_IF;
		7:	IF tx - ta >= tb THEN
				ta := ta + tb;
				tb := multime(time_13 - time_12, M);
				va := value_12;
				vb := value_13;
				temp := value_12;
				state := 8;
			ELSE
				temp := ((vb - va) * TIME_TO_REAL(tx - ta) / TIME_TO_REAL(tb) + va);
			END_IF;
		8:	IF tx - ta >= tb THEN
				temp := value_13;
				run := FALSE;
			ELSE
				temp := ((vb - va) * TIME_TO_REAL(tx - ta) / TIME_TO_REAL(tb) + va);
			END_IF;
	END_CASE;
	Y := temp * K + O;
	ET := tx - t0;
END_IF;

(* revision history
hm	27 feb 2007		rev 1.0
	original version

hm	15. sep2007		rev 1.1
	replaced Time() with T_PLC_MS for compatibility and performance reasons

*)
END_FUNCTION_BLOCK

(* POU engineering/control/FT_IMP, ST *)
FUNCTION_BLOCK FT_IMP
VAR_INPUT
	in : REAL;
	T : TIME;
	K : REAL := 1;
END_VAR
VAR_OUTPUT
	out : REAL;
END_VAR
VAR
	t1 : FT_PT1;
END_VAR

(*
version 1.1	3 Jan 2007
programmer 	hugo
tested by		tobias

FT_IMP is 	an impulse filter (high pass filter) with the time T and factor K.
 
*)
T1(in:= in, T:=T);
out := (in - t1.out) * K;

(*
hm 3.1.2007	rev 1.1
	added factor K

*)
END_FUNCTION_BLOCK

(* POU engineering/control/FT_TN16, ST *)
FUNCTION_BLOCK FT_TN16
VAR_INPUT
	in : REAL;
	T : TIME;
END_VAR
VAR_OUTPUT
	out : REAL;
	trig : BOOL;
END_VAR
VAR
	length : INT := 16;
	X : ARRAY[0..15] OF REAL;
	cnt : INT;
	last : TIME;
	tx: TIME;
	init: BOOL;
END_VAR

(*
version 1.1	16 sep 2007
programmer 	hugo
tested by		tobias

FT_TN16 is delay function, it will delay a signal by a specified time : T and will store 16 values of in before they are put thru to out.
for higher or lower resolution please use FT_TN8 or FT_TN64 instead.
 
*)
(* read system time *)
tx := DWORD_TO_TIME(T_PLC_MS());

trig := FALSE;
IF NOT init THEN
	x[cnt] := in;
	init := TRUE;
	last := tx;
ELSIF tx - last >= T / length THEN
	IF cnt = length - 1 THEN cnt := 0; ELSE cnt := cnt + 1; END_IF;
	Out := X[cnt];
	x[cnt] := in;
	last := tx;
	Trig := TRUE;
END_IF;

(* revision history
hm		1. jan 2007		rev 1.0
	original version

hm		16. sep 2007	rev 1.1
	changes time() to T_plc_ms() for compatibility reasons

*)
END_FUNCTION_BLOCK

(* POU engineering/conversion/length, ST *)
FUNCTION_BLOCK length
VAR_INPUT
	m : REAL;
	p : REAL;
	in : REAL;
	ft : REAL;
	yd : REAL;
	mile : REAL;
	sm : REAL;
	fm : REAL;
END_VAR
VAR_OUTPUT
	Ym : REAL;
	Yp : REAL;
	Yin : REAL;
	Yft : REAL;
	Yyd : REAL;
	Ymile : REAL;
	Ysm : REAL;
	Yfm : REAL;
END_VAR
VAR
END_VAR

(*
version 1.0	27 mar 2007
programmer 	hugo
tested by		oscat

this function converts different length units
any unused input can simply be left open.
different inputs connected at the same time will be added up.

*)
Ym :=	m
		+ p * 0.000376065
		+ in * 0.0254
		+ ft * 0.3048
		+ yd * 0.9144
		+ mile * 1609.344
		+ sm * 1852
		+ fm * 1.829;
Yp := Ym / 0.000376065;
Yin := Ym / 0.0254;
Yft := Ym / 0.3048;
Yyd := Ym / 0.9144;
Ymile := Ym / 1609.344;
Ysm := Ym / 1852;
Yfm := Ym / 1.829;

(*
Länge Meter m SI-Basiseinheit
Astronomische Einheit* AE 1 AE = 149,597 870 · E9 m
Parsec pc 1 pc = 206265 AE = 30,857 · E15 m
Lichtjahr Lj 1 Lj = 9,460 530 · E15 m = 63240 AE = 0,306 59 pc
Ångström Å 1 Å = E–l0 m
typograph. Punkt p 1 p = 0,376 065 mm • im Druckereigewerbe
inch** in 1 in = 2,54 · E–2 m = 25,4 mm***
foot ft 1 ft = 0,3048 m = 30,48 cm
yard yd 1 yd = 0,9144 m
mile mile 1 mile = 1609,344 m
Internat. Seemeile sm 1 sm = 1852 m
Fathom fm 1 fm = 1,829 m • in der Seeschifffahrt

*)
END_FUNCTION_BLOCK

(* POU engineering/control/FT_TN64, ST *)
FUNCTION_BLOCK FT_TN64
VAR_INPUT
	in : REAL;
	T : TIME;
END_VAR
VAR_OUTPUT
	out : REAL;
	trig: BOOL;
END_VAR
VAR
	length : INT := 64;
	X : ARRAY[0..63] OF REAL;
	cnt : INT;
	last : TIME;
	tx: TIME;
	init: BOOL;
END_VAR

(*
version 1.1	15 sep 2007
programmer 	hugo
tested by		tobias

FT_TN7 is delay function, it will delay a signal by a specified time : T and will store 64 values of in before they are put thru to out.
if lower resolution is needed, pls use FT_TN8 or FT_TN16 instead.
 
*)
(* read system time *)
tx := DWORD_TO_TIME(T_PLC_MS());

trig := FALSE;
IF NOT init THEN
	x[cnt] := in;
	init := TRUE;
	last := tx;
ELSIF tx - last >= T / length THEN
	IF cnt = length - 1 THEN cnt := 0; ELSE cnt := cnt + 1; END_IF;
	Out := X[cnt];
	x[cnt] := in;
	last := tx;
	trig := TRUE;
END_IF;

(* revision history
hm		1. jan 2007		rev 1.0
	original version

hm		16. sep 2007	rev 1.1
	changes time() to T_plc_ms() for compatibility reasons

*)
END_FUNCTION_BLOCK

(* POU engineering/control/FT_TN8, ST *)
FUNCTION_BLOCK FT_TN8
VAR_INPUT
	in : REAL;
	T : TIME;
END_VAR
VAR_OUTPUT
	out : REAL;
	trig: BOOL;
END_VAR
VAR
	length : INT := 8;
	X : ARRAY[0..7] OF REAL;
	cnt : INT;
	last : TIME;
	tx: TIME;
	init: BOOL;
END_VAR

(*
version 1.1	15 Sep 2007
programmer 	hugo
tested by		tobias

FT_TN8 is delay function, it will delay a signal by a specified time : T and will store 8 values of in before they are put thru to out.
if higher resolution is needed, pls use FT_TN16 or FT_TN64 instead.
 
*)
tx := DWORD_TO_TIME(T_PLC_MS());
trig := FALSE;
IF NOT init THEN
	x[cnt] := in;
	init := TRUE;
	last := tx;
ELSIF tx - last >= T / length THEN
	IF cnt = length - 1 THEN cnt := 0; ELSE cnt := cnt + 1; END_IF;
	Out := X[cnt];
	x[cnt] := in;
	last := tx;
	trig := TRUE;
END_IF;

(* revision history
hm		1. jan 2007		rev 1.0
	original version

hm		16. sep 2007	rev 1.1
	changes time() to T_plc_ms() for compatibility reasons

*)
END_FUNCTION_BLOCK

(* POU engineering/control/hyst_2, ST *)
FUNCTION_BLOCK hyst_2
VAR_INPUT
	In : REAL;
	val : REAL;
	hys : REAL;
END_VAR
VAR_OUTPUT
	Q : BOOL := 0;
	win: BOOL;
END_VAR
VAR
	X : REAL;
END_VAR


(*
	version 1.0	4 aug 2006
	programmer 	oscat
	tested BY		tobias

this hysteresis function switches the output high if the input signal reaches obove val + hys/2 and will switch to low when the input falls back below val - hys/2 value.
a separate output mid is set if the input stays between low and high value.

*)
X := hys / 2;
IF Q THEN
	IF in < val - x THEN q := FALSE; END_IF;
ELSE
	IF in > val + x THEN q := TRUE; END_IF;
END_IF;
win := in > val - x AND in < val + x;
END_FUNCTION_BLOCK

(* POU engineering/control/Hyst_3, ST *)
FUNCTION_BLOCK Hyst_3
VAR_INPUT
	in : REAL;
	hyst : REAL;
	val1 : REAL;
	val2 : REAL;
END_VAR
VAR_OUTPUT
	Q1 : BOOL;
	Q2 : BOOL;
END_VAR
VAR
END_VAR

(*
	version 1.0	22 jan 2007
	programmer 	oscat
	tested BY		tobias

this is a double hysteresis function. Out1 follows a hysteresis function defined by val1and hyst, while out 2 follows val2 and hyst.
if the input signal is between the two hysteresis switches (val1 and val2) then non of the outputs is active.

*)
IF in < val1 - hyst / 2 THEN
	q1 := TRUE;
ELSIF in > val1 + hyst /2 THEN
	q1 := FALSE;
END_IF;
IF in < val2 - hyst / 2 THEN
	q2 := FALSE;
ELSIF in > val2 + hyst / 2 THEN
	q2 := TRUE;
END_IF;
END_FUNCTION_BLOCK

(* POU engineering/automation/inc_dec, ST *)
FUNCTION_BLOCK inc_dec
VAR_INPUT
	CHa : BOOL;
	CHb : BOOL;
	RST : BOOL := 0;
END_VAR
VAR_OUTPUT
	dir : BOOL;
	cnt : INT;
END_VAR
VAR
	edgea : BOOL := 0;
	clk: BOOL;
	clka: BOOL;
	clkb: BOOL;
	edgeb: BOOL;
	axb: BOOL;
END_VAR

(*
	version 1.0	4 aug 2006
	programmer 	oscat
	tested BY		oscat

incremental decoder with quadruple accuracy.
2 pulses for each channel are created for each directional pulse.
*)
axb := cha XOR chb;

(* create pulses for channel a *)
clka := cha XOR edgea;
edgea := cha;

clkb := chb XOR edgeb;
edgeb := chb;

(* create pulses for both channels *)
clk := clka OR clkb;

(* set the direction output *)
IF axb AND clka THEN dir := TRUE; END_IF;
IF axb AND clkb THEN dir := FALSE; END_IF;

(* increment or decrement the counter *)
IF clk AND dir THEN cnt := cnt + 1; END_IF;
IF clk AND NOT dir THEN cnt := cnt -1; END_IF;

(* reset the counter if rst active *)
IF rst THEN cnt := 0; END_IF;
END_FUNCTION_BLOCK

(* POU engineering/measurements/m_d, ST *)
FUNCTION_BLOCK m_d
VAR_INPUT
	start : BOOL;
	stop : BOOL;
	tmax : TIME := t#10d;
	rst: BOOL;
END_VAR
VAR_OUTPUT
	PT : TIME := t#0ms;
	ET : TIME;
	run : BOOL;
END_VAR
VAR
	edge : BOOL := 0;
	T0 : TIME;
	tx: TIME;
	startup: BOOL;
END_VAR

(*
	version 1.1	16 sep 2007
	programmer 	hugo
	tested BY		tobias

m_d measures the time between a rising edge on start to a rising edge on stop and returs the last measured value on the output PT.
a second output ET is starting from 0 at the rising edge of start and is counting up until the rising edge of stop occurs.
the asynchronous input rst can reset the outputs at any time.
tmax defines a timeout wich is the maximum measurable time between start and stop, if this time is exceeded the outputs will stay at 0.
*)
(* check for rst input *)
IF rst OR et >= tmax THEN
	pt := t#0ms;
	et := t#0ms;
	startup := FALSE;
	run := FALSE;
END_IF;

(* avoid timers to start when input is true at startup *)
IF NOT startup THEN
	edge := start;
	startup := TRUE;
END_IF;

(* read system timer *)
tx := DWORD_TO_TIME(T_PLC_MS());

(* detect rising edge on start *)
IF start AND NOT edge AND NOT stop THEN
	t0 := tx;
	run := TRUE;
	pt := t#0s;
ELSIF stop AND run THEN
	pt := et;
	run := FALSE;
END_IF;
edge := start;
IF run THEN et := tx - t0; END_IF;

(* revision history
hm		2.5.2007	rev 1.0
	original version

hm		16.9.2007	rev 1.1
	changes time() to T_plc_ms() for compatibility reasons

*)
END_FUNCTION_BLOCK

(* POU engineering/measurements/m_tx, ST *)
FUNCTION_BLOCK m_tx
VAR_INPUT
	in: BOOL;
	tmax : TIME := t#10d;
	rst : BOOL;
END_VAR
VAR_OUTPUT
	TH : TIME := t#0ms;
	TL : TIME := t#0ms;
	DC : REAL := 0;
	F: REAL;
	ET : TIME;
END_VAR
VAR
	edge : BOOL := 0;
	start: TIME;
	stop:TIME;
	tx: TIME;
	rise : BOOL;
	fall : BOOL;
	startup: BOOL;
END_VAR

(*
	version 1.2	16 sep 2007
	programmer 	oscat
	tested BY		oscat

this measures the timing of a signal
TH is the high pulse width
TL is the low pulse width
DC is the duty cycle
F is the frequency
ET will start at 0 with a rising edge and count up till the next rising edge starts from 0 again. 
the acuracy depends on the cycle time of the sps and is limited to 1ms resolution.
an asynchronous reset can reset all outputs to 0 at any time.
the input tmax can configure a timeout for ET where the function block will outomatically reset itself.
tmx is predefined to 10 days.
*)
(* check FOR rst input *)
IF rst OR (et >= tmax) THEN
	rise := FALSE;
	fall := FALSE;
	startup := FALSE;
	th := t#0ms;
	tl := t#0ms;
	DC := 0;
	F := 0;
	ET := t#0s;
END_IF;

(* avoid timers to start when input is true at startup *)
IF NOT startup THEN
	edge := in;
	startup := TRUE;
END_IF;

(* read system timer *)
tx := DWORD_TO_TIME(T_PLC_MS());

(* edge trigger rising and falling edge *)
IF in XOR edge THEN
	edge := in;
	(* rising edge starts measurement *)
	IF in THEN
		start := Tx;
		rise := TRUE;
		IF fall THEN tl := start - stop; END_IF;
		IF th > t#0ms AND tl > t#0ms THEN
			dc := TIME_TO_REAL(th) / TIME_TO_REAL(th+tl);
			f := 1000 / TIME_TO_REAL(th + tl);
		END_IF;
	(* falling edge starts second cycle measurement *)
	ELSE
		stop := Tx;
		fall := TRUE;
		IF rise THEN th := stop - start; END_IF;
		IF th > t#0ms AND tl > t#0ms THEN
			dc := TIME_TO_REAL(th) /  TIME_TO_REAL(th+tl);
			f := 1000 / TIME_TO_REAL(th + tl);
		END_IF;
	END_IF;
END_IF;
IF rise THEN et := tx - start; END_IF;

(* revision history
hm		4. aug 2006	rev 1.0
	original version

hm		2. mai 2007	rev 1.1
	made sure that no undefined values would be measured at startup conditions
	added output et
	added rst input
	added tmax input

hm		16.9.2007	rev 1.2
	changes time() to T_plc_ms() for compatibility reasons

*)
END_FUNCTION_BLOCK

(* POU engineering/signal generators/gen_rdm, ST *)
FUNCTION_BLOCK gen_rdm
VAR_INPUT
	PT : TIME;
	AM : REAL := 1;
	OS : REAL;
END_VAR
VAR_OUTPUT
	Q : BOOL;
	Out : REAL;
END_VAR
VAR
	tx : TIME;
	last : TIME;
	init : BOOL;
END_VAR

(*
	version 1.1	16 sep 2007
	programmer 	oscat
	tested BY		oscat

this signal generator generates a random output. The signal is defined by period time (PT), 
amplitude (AM), offset (OS).
The Output waveform will have its max peak at AM/2 + OS and its minimum peak at -AM/2 + OS. 
The period time PT defines how often the output signal will jump to a new randow value.
The Output Q will be true for one cycle anytime the output OUT has changed

*)
(* read system time and prepare input data *)
tx := DWORD_TO_TIME(T_PLC_MS()) - last;

(* init section *)
IF NOT init THEN
	init := TRUE;
	last := tx;
	tx := t#0s;
END_IF;

(* add last if one cycle is finished *)
IF tx >= pt THEN
	last := last + pt;
	tx := tx - pt;

	(* generate output signal *)
	out := am * (RDM(0) - 0.5) + os;
	q := TRUE;
ELSE
	q := FALSE;
END_IF;

(* revision history

hm	7.2.2007		rev 1.0
	original version

hm	16.9.2007		rev 1.1
	changes time() to T_plc_ms() for compatibility reasons

*)
END_FUNCTION_BLOCK

(* POU engineering/signal generators/gen_rmp, ST *)
FUNCTION_BLOCK gen_rmp
VAR_INPUT
	PT : TIME := t#1s;
	AM : REAL := 1;
	OS : REAL := 0;
	DL : REAL := 0;
END_VAR
VAR_OUTPUT
	Q : BOOL;
	Out : REAL;
END_VAR
VAR
	tx : TIME;
	last : TIME;
	init : BOOL;
	temp : REAL;
	ltemp: REAL;
END_VAR

(*
	version 1.1	17 sep 2007
	programmer 	oscat
	tested BY		oscat

this signal generator generates a ramp wave output. The ramp wave signal is defined by period time (PT), 
amplitude (AM), offset (OS) and a specific delay for the output signal (DL).
The Output waveform will have its minimum peak at OS and its maximum peak at AM + OS. 
The delay input can delay a signal up to PT, this can be useful to synchronize different generators 
and generate interleaving signals.
in addition to the analog output Out there is a second boolean output Q with is true for one cycle when the ramp starts.
*)
(* read system time and prepare input data *)
tx := DWORD_TO_TIME(T_PLC_MS()) - last;
DL := modR(dl,1);
IF dl < 0 THEN dl := 1 - dl; END_IF;

(* init section *)
IF NOT init THEN
	init := TRUE;
	last := tx;
	tx := t#0s;
END_IF;

(* add last if one cycle is finished *)
IF tx >= pt THEN
	last := last + pt;
	tx := tx - pt;
END_IF;

(* generate sine wave *)
ltemp := temp;
temp := fract(TIME_TO_REAL(tx + multime(pt, dl)) / TIME_TO_REAL(pt));
out := am * temp + os;

(* boolean output Q *)
IF temp < ltemp THEN
	q := TRUE;
ELSE
	q := FALSE;
END_IF;

(* revision history
hm	3. mar 2007		rev 1.0
	original version

hm	17 sep 2007		rev 1.1
	replaced time() with t_plc_ms for compatibilitx reasons

*)
END_FUNCTION_BLOCK

(* POU engineering/signal generators/gen_sin, ST *)
FUNCTION_BLOCK gen_sin
VAR_INPUT
	PT : TIME;
	AM : REAL := 1;
	OS : REAL;
	DL : REAL;
END_VAR
VAR_OUTPUT
	Q : BOOL;
	Out : REAL;
END_VAR
VAR
	tx : TIME;
	last : TIME;
	init : BOOL;
	temp : REAL;
END_VAR

(*
	version 1.1	17 sep 2007
	programmer 	oscat
	tested BY		oscat

this signal generator generates a sine wave output. The sine wave signal is defined by period time (PT), 
amplitude (AM), offset (OS) and a specific delay for the output signal (DL).
The Output waveform will have its max peak at AM/2 + OS and its minimum peak at -AM/2 + OS. 
The delay input can delay a signal up to PT, this can be useful to synchronize different generators 
and generate interleaving signals. A Cos wave can be generated accordingly.
in addition to a analog output Out there is a second boolean output Q with the corresponding binary signal.
*)
(* read system time and prepare input data *)
tx := DWORD_TO_TIME(T_PLC_MS()) - last;
DL := modR(dl,1);
IF dl < 0 THEN dl := 1 - dl; END_IF;

(* init section *)
IF NOT init THEN
	init := TRUE;
	last := tx;
	tx := t#0s;
END_IF;

(* add last if one cycle is finished *)
IF tx >= pt THEN
	last := last + pt;
	tx := tx - pt;
END_IF;

(* generate sine wave *)
temp := SIN(PI2 * TIME_TO_DWORD(tx + multime(pt, dl)) / TIME_TO_DWORD(pt));
out := am / 2 *  temp + os;

(* boolean output Q *)
q := NOT sign_R(temp);

(* revision history
hm	22. jan 2007		rev 1.0
	original version

hm	17 sep 2007		rev 1.1
	replaced time() with t_plc_ms for compatibilitx reasons

*)
END_FUNCTION_BLOCK

(* POU engineering/signal generators/gen_sqr, ST *)
FUNCTION_BLOCK gen_sqr
VAR_INPUT
	PT : TIME;
	AM : REAL;
	OS : REAL;
	DC : REAL := 0.5;
	DL : REAL;
END_VAR
VAR_OUTPUT
	Q : BOOL;
	Out : REAL;
END_VAR
VAR
	tx : TIME;
	last : TIME;
	init: BOOL;
END_VAR

(*
	version 1.2	17 sep 2007
	programmer 	oscat
	tested BY		oscat

this signal generator generates a square wave output. The square wave signal is defined by period time (PT), 
amplitude (AM), offset (OS), duty cycle (DC) and a specific delay for the output signal (DL).
The Output waveform will switch between AM/2 + OS and -AM/2 + OS. The DC input specifies ther duty cycle, 
DC = 0 means output is low at all times and 1 means output is high at all times.
The delay input can delay a signal up to PT, this can be useful to synchronize different generators and generate interleaving signals.
in addition to a analog output Out there is a second boolean output Q.
*)
(* check dc = 1 or 0 *)
IF dc = 0 THEN
	out := am / -2 + os;
	Q := FALSE;
	RETURN;
ELSIF dc = 1 THEN
	out := am /2 + os;
	Q := TRUE;
	RETURN;
END_IF;

(* read system time and prepare input data *)
tx := DWORD_TO_TIME(T_PLC_MS()) - last;
DL := modR(dl,1);
IF dl < 0 THEN dl := 1 - dl; END_IF;
dc := modR(dc,1);
IF dc < 0 THEN dc := 1 - dc; END_IF;

(* init section *)
IF NOT init THEN
	init := TRUE;
	last := tx;
	tx := t#0s;
END_IF;

(* add last if one cycle is finished *)
IF tx >= pt THEN
	last := last + pt;
	tx := tx - pt;
END_IF;

(* check if falling or rising edge first *)
IF multime(pt, dl + dc) >= pt THEN
	(* generate falling edge *)
	IF tx >= multime(pt, dl + dc - 1) THEN
		out := am / -2 + os;
		Q := FALSE;
	END_IF;
	(* generate rising edge *)
	IF tx >= multime(pt, dl) THEN
		out := am / 2 + os;
		Q := TRUE;
	END_IF;
ELSE
	(* generate rising edge first *)
	IF tx >= multime(pt, dl) THEN
		out := am / 2 + os;
		Q := TRUE;
	END_IF;
	(* generate falling edge *)
	IF tx >= multime(pt, dl + dc) THEN
		out := am / -2 +os;
		Q := FALSE;
	END_IF;
END_IF;

(* revision history

hm	12. feb 2007	rev 1.1
	added default value for dc = 0.5

hm	17 sep 2007		rev 1.2
	replaced time() with t_plc_ms for compatibilitx reasons


*)
END_FUNCTION_BLOCK

(* POU engineering/signal generators/pwm_dc, ST *)
FUNCTION_BLOCK pwm_dc
VAR_INPUT
	F : REAL;
	DC : REAL;
END_VAR
VAR_OUTPUT
	Q : BOOL;
END_VAR
VAR
	clk: CLK_Prg;
	pulse: TP_R;
END_VAR

(*
	version 1.1	25 feb 2007
	programmer 	oscat
	tested BY		oscat

this signal generator generates a square wave signal which is specified by the frequency and the duty cycle
*)
CLK(PT := REAL_TO_TIME(1000/F));
Pulse(in := clk.Q, pt := REAL_TO_TIME(1000/F*DC));
Q := pulse.Q;

(* revision history

hm		25. feb 2007	rev 1.1
	recoded in st for better performance and better portability

*)
END_FUNCTION_BLOCK

(* POU Logic/generators/TP_R, ST *)
FUNCTION_BLOCK TP_R
VAR_INPUT
	in : BOOL;
	PT : TIME;
END_VAR
VAR_OUTPUT
	Q : BOOL := 0;
	ET : TIME := t#0ms;
END_VAR
VAR
	edge : BOOL := FALSE;
	start : TIME := t#0ms;
	tx: TIME;
END_VAR

(*
version 1.1	17 sep 2007
programmer 	hugo
tested by		tobias

retriggerable edge triggered pulse similar to TP but with a retrigger function
if the pt input is 0 then output is always low.
*)
(* read system_time *)
tx := DWORD_TO_TIME(T_PLC_MS());

(* rising edge trigger *)
IF in AND NOT edge THEN
	start := Tx;
	IF pt > t#0ms THEN Q := TRUE; END_IF;
END_IF;
edge := in;
IF q THEN
	et := Tx - start;
	IF et >= PT THEN
		Q := FALSE;
		et := t#0ms;
	END_IF;
END_IF;


(* revision history
hm	4. aug 2006		rev 1.0
	original version

hm	17. sep 2007	rev 1.1
	replaced time() with T_PLC_MS() for compatibility reasons
	
*)
END_FUNCTION_BLOCK

(* POU engineering/signal generators/pwm_pw, ST *)
FUNCTION_BLOCK pwm_pw
VAR_INPUT
	F : REAL;
	PW : TIME;
END_VAR
VAR_OUTPUT
	Q : BOOL;
END_VAR
VAR
	clk: CLK_Prg;
	pulse: TP_R;
END_VAR

(*
	version 1.1	25 feb 2007
	programmer 	oscat
	tested BY		oscat

this signal generator generates a square wave signal which is specified by the frequency and the pulse width.
*)
CLK(PT := REAL_TO_TIME(1000/F));
Pulse(in := clk.Q, pt := pw);
Q := pulse.Q;

(* revision history

hm		25. feb 2007	rev 1.1
	recoded in st for better performance and better portability

*)
END_FUNCTION_BLOCK

(* POU engineering/signal generators/rmp_soft, ST *)
FUNCTION_BLOCK rmp_soft
VAR_INPUT
	IN : BOOL;
	val : BYTE;
END_VAR
VAR_INPUT CONSTANT
	pt_on: TIME := T#100ms;
	PT_off : TIME := T#100ms;
END_VAR
VAR CONSTANT
	steps : INT := 255;
END_VAR
VAR_OUTPUT
	Out : BYTE := 0;
END_VAR
VAR
	last_step : TIME := T#0ms;
	now : TIME;
	x :REAL := 0;
END_VAR

(*
	version 1.2	17 sep 2007
	programmer 	oscat
	tested BY		oscat

this soft on/off ramp generator generates a soft on and soft off ramp while the max on value is set by the input
the time for a full ramp can be set by config variables for up and down ramp.
*)
(* read system time *)
now := DWORD_TO_TIME(T_PLC_MS());

IF in  AND out < val THEN
	(* generate on ramp *)
	x := out + TIME_TO_REAL(now -last_step)*steps/TIME_TO_REAL(pt_on);
	IF x > val THEN
		out := val;
		x := val;
	ELSE out := REAL_TO_BYTE(x); END_IF;
	last_step := now;
ELSIF NOT in AND out > 0 THEN
	(* generate off ramp *)
	x := out - TIME_TO_REAL(now - last_step)*steps/TIME_TO_REAL(pt_off);
	IF x  < 0 THEN
		out := 0;
		x := 0;
	ELSE out := REAL_TO_BYTE(x); END_IF;
	last_step := now;
ELSIF in AND out > val THEN
	(* generate ramp down to input value *)
	x := out - TIME_TO_REAL(now - last_step)*steps/TIME_TO_REAL(pt_off);
	IF x  < val THEN
		out := val;
		x := val;
	ELSE out := REAL_TO_BYTE(x); END_IF;
	last_step := now;
END_IF;
IF out = val OR out = 0 THEN last_step := now; END_IF;


(* revision history

hm 22.1.2007	rev 1.1
	deleted unused variables X1 and I, X2 and X3

hm	17.9.2007	rev 1.2
	replaced time() with t_plc_ms() for compatibility reasons

*)
END_FUNCTION_BLOCK

(* POU engineering/signal processing/SH, ST *)
FUNCTION_BLOCK SH
VAR_INPUT
	in : REAL;
	CLK : BOOL;
END_VAR
VAR_OUTPUT
	out : REAL;
	trig : BOOL;
END_VAR
VAR
	edge : BOOL;
END_VAR

(*
version 1.1	16 jan 2007
programmer 	hugo
tested by		tobias

this sample and hold module samples an input at the rising edge of clk an stores it in out.
the out stays stable until the next rising clk edge appears.
a trigger output as active for one cycle when the output was updated.

*)
IF clk AND NOT edge THEN
	out := in;
	trig := TRUE;
ELSE;
	trig := FALSE;
END_IF;
edge := clk;

(* revision history

hm 16.1.2007	rev 1.1
	added trig output

*)
END_FUNCTION_BLOCK

(* POU engineering/signal processing/SH_1, ST *)
FUNCTION_BLOCK SH_1
VAR_INPUT
	in : REAL;
	PT : TIME;
END_VAR
VAR_OUTPUT
	out : REAL;
	Trig : BOOL;
END_VAR
VAR
	last : TIME;
	tx: TIME;
END_VAR

(*
version 1.2	17 sep 2007
programmer 	hugo
tested by		tobias

this sample and hold module samples an input every PT seconds.
after a ample is taken the output Trig will be active for one cycle.

*)
(* read system time *)
tx := DWORD_TO_TIME(T_PLC_MS());

IF tx - last >= PT THEN
	last := tx;
	out := in;
	trig := TRUE;
ELSE
	trig := FALSE;
END_IF;

(* revision history

HM	6.1.2007	rev 1.1
	added trig output

HM	17.9.2007	rev 1.2
	replaced time() with T_PLC_MS() for compatibility reasons
*)
END_FUNCTION_BLOCK

(* POU engineering/signal processing/SH_2, ST *)
FUNCTION_BLOCK SH_2
VAR_INPUT
	in : REAL;
	PT : TIME;
	N : INT;
	disc : INT;
END_VAR
VAR_OUTPUT
	out : REAL;
	trig : BOOL;
	avg : REAL;
	high: REAL;
	low: REAL;
END_VAR
VAR
	M : INT;
	buf : ARRAY[0..15] OF REAL;
	buf2 : ARRAY[0..15] OF REAL;
	last : TIME;
	i : INT;
	start: INT;
	temp: REAL;
	stop: INT;
	tx: TIME;
END_VAR

(*
version 1.3	17 sep 2007
programmer 	hugo
tested by		tobias

this sample and hold module samples an input every PT seconds.
this sample and hold also does avg and other calculations with the input data.
an average is calculated over N samples while for this calculation disc samples are discarded,
disc = 0 all samples are averaged,
if disc = 1 the lowest value is ignored,
if disc = 2 the lowest and highest values are ignored, 
and so on.....

*)
(* read system time *)
tx := DWORD_TO_TIME(T_PLC_MS());

IF tx - last >= PT THEN
	last := tx;
	trig := TRUE;

	(* limit M to 0..16 *)
	M := LIMIT(1,N,16);

	(* edge detected lets take the sample *)
	FOR i := M - 1 TO 1 BY -1 DO buf2[i] := buf2[i-1]; END_FOR;
	buf2[0] := in;
	out := in;
	buf := buf2;

	(* sort the ARRAY lowest value AT 0 *)
	FOR start := 0 TO M - 2 DO
		FOR i := start+1 TO M - 1 DO
			IF buf[start] > buf[i] THEN
				temp := buf[start];
				buf[start] := buf[i];
				buf[i] := temp;
			END_IF;
		END_FOR;
	END_FOR;

	(* any calculation with the samples is here *)
	stop := M - 1 - disc / 2;
	start := 0 + disc / 2;
	IF NOT even(disc) THEN start := start + 1; END_IF;
	avg := 0;
	FOR i := start TO stop DO avg := avg + buf[i]; END_FOR;
	avg := avg / (stop - start +1);
	low := buf[start];
	high := buf[stop];
ELSE
	Trig := FALSE;
END_IF;

(* revision history
hm 20.1.2007	rev 1.1
	added input N to specify the amout of samples for average and high low calculations
	added trig output

hm 10.9.2007 rev 1.2
	an error would be generated if N was set to 0, now n is forced to1 if set to 0.
	index was out of array.

hm	17.9.2007	rev 1.3
	replaced time() with t_plc_ms() for compatibility reasons

*)
END_FUNCTION_BLOCK

(* POU engineering/signal processing/SH_T, ST *)
FUNCTION_BLOCK SH_T
VAR_INPUT
	in : REAL;
	EN : BOOL;
END_VAR
VAR_OUTPUT
	out : REAL;
END_VAR
VAR
END_VAR

(*
version 1.0	1 sep 2006
programmer 	hugo
tested by		tobias

this sample and hold module samples an input while en is high.
during the high time of en the output follows in.
the out stays stable until the en goes high again.
*)
IF en THEN out := in; END_IF;
END_FUNCTION_BLOCK

(* POU engineering/signal processing/stair2, ST *)
FUNCTION_BLOCK stair2
VAR_INPUT
	X : REAL;
	D : REAL;
END_VAR
VAR_OUTPUT
	Y: REAL;
END_VAR
VAR_TEMP
	tmp : REAL;
END_VAR


(*
version 1.0	28 jan 2007
programmer 	oscat
tested by		tobias

the function stair2 converts an anlog input signal to a staircase like output.
D is the step width for the output signal. the output will use D as a hysteresis for a stairchange.
if D = 0 then the output follows the input without a chage.
*) 
tmp := TRUNC(X / D);

IF X >= Y AND X >= 0 THEN
	Y := TRUNC(X / D) * D;
ELSIF X < Y AND X >= 0 THEN
	Y := (TRUNC(X/d) + 1) * D;
ELSIF X >= Y AND X < 0 THEN
	Y := (TRUNC(X/D)-1) * D;
ELSIF X < Y AND X < 0 THEN
	Y := TRUNC(X/D) *D;
END_IF;
END_FUNCTION_BLOCK

(* POU Logic/FF edge triggered/FF_D2E, ST *)
FUNCTION_BLOCK FF_D2E
VAR_INPUT
	D0 : BOOL := 0;
	D1 : BOOL := 0;
	CLK : BOOL;
	RST : BOOL := 0;
END_VAR
VAR_OUTPUT
	Q0 : BOOL := 0;
	Q1 : BOOL := 0;
END_VAR
VAR
	edge : BOOL;
END_VAR

(*
version 1.0	4 aug 2006
programmer 	hugo
tested by		tobias

dual D-type flip flop with reset and rising clock trigger

executioin TIME on wago 750-841 = 6us
*)
IF rst THEN
	Q0 := FALSE;
	Q1 := FALSE;
ELSE
	IF clk AND NOT edge THEN
		Q0 := D0;
		Q1 := D1;
	END_IF;
END_IF;
edge := CLK;
END_FUNCTION_BLOCK

